(* CODESYS project uninc.library
   Company: Beckhoff Automation GmbH & Co. KG
   DefaultNamespace: TC3_UniNC
   Version: 1.0.6.2
   Placeholder: UniNc Gruppe 11
   Author: Bernhard Edenfeld, Benedikt Daut, Christian Frickenstein
   Description: FBs für die Nutzung der NC, Sercos-Achsen, Encoder-Achsen und Eil-Schleichachsen im Stil der Gruppe 11
   Title: UniNc Gruppe 11

Project tree, tasks and I/O mapping:
  libraries: Tc2_MC2, * (Beckhoff Automation GmbH); Tc2_MC2_Drive, * (Beckhoff Automation GmbH); Tc2_Standard, * (Beckhoff Automation GmbH); Tc2_System, * (Beckhoff Automation GmbH); UniLib Gruppe 11, * (Beckhoff Automation GmbH & Co. KG)
  DUTs/
    data type E_AchsFahrauftraege
    data type ST_DiagAxis
    data type ST_UniEinschleifen
  GVLs/
    global variables GlobalVar_NC
    global variables NcParameter
  POUs/
    function block FB_AchsKontrlAnstg [ST]: a_AchsStatus, b_AchsParam, c_AchsFreigb, d_AchsReferz, e_AchsHdFkt, f_AchsKopplg, g_AchsAuftrg, h_AchsEndlos, i_AchsModulo, k_AchsReset, x_AchsMeldg
    function block FB_AchsStartAusf [ST]
    function block FB_Bremsentest_BremseEinschleifen [ST]: a_Error, a_LogZeile, b_AnwEinschleifen
    function block FB_BremsentestMitLog [ST]: a_Error, a_LogZeile
    function block FB_BremsentestMitLog_FW07 [ST]: a_Error, a_LogZeile
    function block FB_CtrlXGrupEinschalt [ST]
  VISUs/
    Intern/
      visualisation V_DiagAchse
  text list GlobalTextList
*)

// DUTs/E_AchsFahrauftraege
{attribute 'qualified_only'}
{attribute 'strict'}
TYPE E_AchsFahrauftraege :
(
	eKoppelPosition 			:= 1,	// Index für arrPTP_start[]: Achse fährt eine Korrekturposition an um mit einer Masterachse zu koppeln mit 5% der Max-Geschwindigkeit
	eGrundPosition				:= 2,	// Index für arrPTP_start[]: Achse fährt die Grundposition aus den Parametern an mit 25% der Max-Geschwindigkeit
	eBearbeitungsPosition	:= 3	// Index für arrPTP_start[]: Achse fährt zur Bearbeitungsposition aus den Zielvorgaben an mit der prozentual gewählten Zielgeschwindigkeit
);
END_TYPE

// DUTs/ST_DiagAxis
TYPE ST_DiagAxis :
STRUCT
	nAcutalLength	: UINT;	// Tatsächliche länge der Meldung
	nMaxLength		: UINT;	// Maximal mögliche länge der Meldung 
	sDiagMessage	: T_MaxString;	// Standardlänge der Meldung. Kann aber beschränkt ausgelesen werden durch nAcutalLength.
END_STRUCT
END_TYPE

// DUTs/ST_UniEinschleifen
// Struktur für eine standardisierte Grundstellungsanwahl mit einer HMI-Taste und Meldungen 
{attribute 'pack_mode' := '1'}
TYPE ST_UniEinschleifen :
STRUCT
// Eine Handfunktionstaste für die Grundstellungsfahrt.
{attribute 'MaschPara.Name' := 'Handfunktion:'}	// Das Array ist Teil der Handfunktionen und wird mit 'Handfunktion:' betitelt
{attribute 'MaschPara.Handfunktion.Btn1' := '1 TextHandFkt'} // Handfunktion.Btn[X] ist der Taster im Array. TextHandFkt ist default Text, wenn z.B. die PLC nicht läuft
	stHandFktHMI		: ARRAY [1..1] OF ST_HandFktHMI;

END_STRUCT
END_TYPE

// GVLs/GlobalVar_NC
{attribute 'Tc2GvlVarNames'}
VAR_GLOBAL
	arrStartAusf							:ARRAY[0..cAnzAchsen] OF FB_AchsStartAusf;	// Vorschlag für eine allgemeine Instanz: Achsstart-FB für alle Achsen vordefiniert. Kann im Projekt aufgerufen werden. 

	arrNcAchsReset							:ARRAY[0..cAnzAchsen] OF BOOL;	// Vorschlag für eine allgemeine Variable: NC-AchsReset für eine bestimmte Achse 
	
	arrAchsDiag								:ARRAY[0..cAnzAchsen] OF Tc2_System.T_MaxString;	// Diagnose/Zustand der SoE-Achsen. S-0-0095
	
	// Allgemeine Achsvariablen
	bNcAchsResetErfordl					:BOOL;	// Vorschlag für eine allgemeine Variable: mindestens eine NC-Achse hat einen Fehler und ein Reset ist erforderlich.
	bAchsFreifahrErfordl					:BOOL;	// Vorschlag für eine allgemeine Variable: mindestens eine Achse hat oder hatte die Endlagen angefahren und muss von dieser manuell heruntergefahren werden
	bAchsRestartErfordl					:BOOL;	// Vorschlag für eine allgemeine Variable:
	bNcAchsResetAngw						:BOOL;	// Vorschlag für eine allgemeine Variable: NC-Reset wurde durch Bediener angewählt
	bAchsFreifahrAngw						:BOOL;	// Vorschlag für eine allgemeine Variable: Achsen Freifahren wurde durch Bediener angewählt
	bAntriebResetAktiv					:BOOL;	// Vorschlag für eine allgemeine Variable: Hardware-Reset ist aktiv
	
	// Override
	fOverridePTP							:LREAL:= 100;	// Vordefinierter maximaler Override für alle Achsen
END_VAR
VAR_GLOBAL CONSTANT
	// Fahraufträge Achsen
	cKopplPos	: INT:= 1;	// Index für arrPTP_start[]: Achse fährt eine Korrekturposition an um mit einer Masterachse zu koppeln mit 5% der Max-Geschwindigkeit
	cGrundPos	: INT:= 2;	// Index für arrPTP_start[]: Achse fährt die Grundposition aus den Parametern an mit 25% der Max-Geschwindigkeit
	cBearbPos	: INT:= 3;	// Index für arrPTP_start[]: Achse fährt zur Bearbeitungsposition aus den Zielvorgaben an mit der prozentual gewählten Zielgeschwindigkeit
END_VAR

// GVLs/NcParameter
{attribute 'Tc2GvlVarNames'}
VAR_GLOBAL CONSTANT
	// Gesamtanzahl Achsen
	cAnzAchsen			: INT:= 100;	// Achsen mit Encoder und Drive. Also auch Eil-Schleichachsen und Encoderachsen
	cAnzAchsenReal		: INT:= 8;	// Nur Achsen mit Drive. Also SoE und Eil-Schleichachsen
END_VAR

// POUs/FB_AchsKontrlAnstg
(*
Beschreibung :	Allg. Achshändling (MC2-Lib)
					Datentypen: Struct_NcAchsen
TwinCat Vers.:	3.1.4024.25							
Erstellt		 :	Anlagentechnik Grp.11 (BECKHOFF AUTOMATION)
*)
FUNCTION_BLOCK FB_AchsKontrlAnstg
VAR_IN_OUT
	IQ_stAchse						: TC3_UniLib.ST_NcAchsen;
	IQ_fbAxisRef					: Tc2_MC2.AXIS_REF;
END_VAR
VAR_INPUT
	I_refNcAchsen					: REFERENCE TO ARRAY [1..cAnzAchsen] OF Tc2_MC2.AXIS_REF;
	I_nBetrArt						: INT	:= 0;		(*0:Standard-PTP/1:Endlosbetrieb/2:Modulobetrieb *)
	I_fOverride						: LREAL := 100;	// Override für diese Achse, bei Nichtverwendung 100%
	I_bEndlagenExtern				: BOOL;
	I_bAutoStopAktiv				: BOOL := TRUE;
{attribute 'hide'}	
	I_eRichtungModulo				: MC_Direction := MC_Positive_Direction;
END_VAR
VAR_OUTPUT
END_VAR
VAR
	(*a_AchsStatus*)
	tonHwFehler			:Tc2_Standard.TON;
	stDiagAxis			:ST_DiagAxis;
	nIdn					:WORD;

	(*b_AchsParam*)
	fbAchsPar1L			:Tc2_MC2.MC_ReadParameter;
	stAchsPar1LOut		:Tc2_MC2.ST_McOutputs;
	fbAchsPar2L			:Tc2_MC2.MC_ReadParameter;
	stAchsPar2LOut		:Tc2_MC2.ST_McOutputs;
	fbAchsPar3L			:Tc2_MC2.MC_ReadBoolParameter;
	stAchsPar3LOut		:Tc2_MC2.ST_McOutputs;
	fbAchsPar4L			:Tc2_MC2.MC_ReadBoolParameter;
	stAchsPar4LOut		:Tc2_MC2.ST_McOutputs;
	fbAchsPar5L			:Tc2_MC2.MC_ReadParameter;
	stAchsPar5LOut		:Tc2_MC2.ST_McOutputs;
	fbAchsPar1S			:Tc2_MC2.MC_WriteParameter;
	stAchsPar1SOut		:Tc2_MC2.ST_McOutputs;
	fbAchsPar2S			:Tc2_MC2.MC_WriteParameter;
	stAchsPar2SOut		:Tc2_MC2.ST_McOutputs;
	
	fbAchsParName		:Tc2_MC2.MC_ReadParameterSet;
	stAchsParSet		:Tc2_MC2.ST_AxisParameterSet;
	stAchsParName		:Tc2_MC2.ST_McOutputs;

	rtrigParamLesZykl	:Tc2_Standard.R_TRIG;
	bEndlMinLes			:BOOL;
	bEndlMinSchr		:BOOL;
	fEndlBegrMin		:LREAL;
	bEndlMaxLes			:BOOL;
	bEndlMaxSchr		:BOOL;
	fEndlBegrMax		:LREAL;

	(*c_AchsFreigb*)
	fbAchsFreig			:Tc2_MC2.MC_Power;
	stAchsFreigOut		:Tc2_MC2.ST_McOutputs;

	tonVerzVorschFrg	:Tc2_Standard.TON;
	tonVerzEndlgStop	:Tc2_Standard.TON;
	tonVerzAntrbFehl	:Tc2_Standard.TON;

	(*d_AchsReferz*)
	fbAchsReferenz		:Tc2_MC2.MC_Home;
	stAchsReferenzOut	:Tc2_MC2.ST_McOutputs;
	fbAchsIstwSetz		:Tc2_MC2.MC_SetPosition;
	stAchsIstwSetzOut	:Tc2_MC2.ST_McOutputs;

	(*e_AchsHdFkt*)
	fbAchsHandfkt		:Tc2_MC2.MC_Jog;
	stAchsHandfktOut	:Tc2_MC2.ST_McOutputs;

	(*f_AchsKopplg*)
	fbAchsAnkoppln		:Tc2_MC2.MC_GearInDyn;
	stAchsAnkopplnOut	:Tc2_MC2.ST_McOutputs;
	fbAchsAbkoppln		:Tc2_MC2.MC_GearOut;
	stAchsAbkopplnOut	:Tc2_MC2.ST_McOutputs;

	(*g_AchsAuftrg*)
	fbAchsStartA1		:Tc2_MC2.MC_MoveAbsolute; (*Standard*)
	fbAchsStartA2		:Tc2_MC2.MC_MoveVelocity; (*Endlos*)
	fbAchsStartA3		:Tc2_MC2.MC_MoveModulo; (*Modulo*)
	stAchsStartAOut	:Tc2_MC2.ST_McOutputs;
	fbAchsStartB1		:Tc2_MC2.MC_MoveAbsolute; (*Standard*)
	fbAchsStartB2		:Tc2_MC2.MC_MoveVelocity; (*Endlos*)
	fbAchsStartB3		:Tc2_MC2.MC_MoveModulo; (*Modulo*)
	stAchsStartBOut	:Tc2_MC2.ST_McOutputs;
	fbAchsStop			:Tc2_MC2.MC_Halt;
	stAchsStopOut		:Tc2_MC2.ST_McOutputs;

	fAuftrZielPos		:LREAL;
	fLetztZielPos		:LREAL;
	fAuftrGeschw		:LREAL;
	fLetztGeschw		:LREAL;
	nAuftrBuffMode		:Tc2_MC2.MC_BufferMode;
	bAuftrStart			:BOOL;
	nAuftrState			:INT;
	bNeuAuftrVorg		:BOOL;
	bAuftrStartA		:BOOL;
	bAuftrAktivA		:BOOL;
	bAuftrFertigA		:BOOL;
	bAuftrStartB		:BOOL;
	bAuftrAktivB		:BOOL;
	bAuftrFertigB		:BOOL;
	bAuftrStop			:BOOL;
	bAuftrGestoppt		:BOOL;
	fAuftrOverride		:LREAL;
	tonAuftrLfZeit		:Tc2_Standard.TON;

	(*k_AchsReset*)
	tpReset				:Tc2_Standard.TP;
	bInit					:BOOL;
	fbAchsReset			:Tc2_MC2.MC_Reset;
	stAchsResetOut		:Tc2_MC2.ST_McOutputs;

	(*x_AchsMeldg*)
	nAchsMeldNr			:INT;
	fbDiagMessages		:FB_SoERead;
END_VAR

	(*Achs-Kontrollfkt./-Ansteuerung*)
	
	(**************************************************)	

	a_AchsStatus();	(*Achsstatus lesen/sotieren*)
							(*Achsenistwert lesen*)

	(**************************************************)	

	b_AchsParam();		(*Achsparameter lesen*)
							(*Achsparameter schreiben*)

	(**************************************************)	

	c_AchsFreigb();	(*Achsfreigaben ermitteln*)
							(*Achsfreigaben schreiben*)

	(**************************************************)	

	d_AchsReferz();	(*Achse referieren*)
							(*Achsistwert setzen*)

	(**************************************************)	

	e_AchsHdFkt();		(*Achshandfunktionen*)

	(**************************************************)	

	f_AchsKopplg();	(*Achse an.-abkoppeln*)

	(**************************************************)	

	CASE I_nBetrArt OF
0:	g_AchsAuftrg();	(*Achswerte schreiben / Achse starten / Achse stoppen*)
1:	h_AchsEndlos();	(*			0:Standard-PTP / 1:Endlosbetrieb /2:Modulobetrieb            *)
2:	i_AchsModulo();	(*			0:Standard-PTP / 1:Endlosbetrieb /2:Modulobetrieb            *)
	END_CASE

	(**************************************************)	

	k_AchsReset();		(*Achse zurücksetzen*)

	(**************************************************)	

	x_AchsMeldg();		(*Achsmeldungen ausgeben*)

	(**************************************************)

ACTION a_AchsStatus:
	// Achsstatus lesen/sotieren
	IQ_fbAxisRef.ReadStatus();
	IQ_stAchse.nAxNr						:= TO_INT(IQ_fbAxisRef.NcToPlc.AxisId);

	IQ_stAchse.bNcFehler					:= IQ_fbAxisRef.Status.Error;
	IQ_stAchse.nFehlerNr					:= IQ_fbAxisRef.Status.ErrorID;
	IQ_stAchse.bBetrbBer					:= IQ_fbAxisRef.Status.Operational;

	IQ_stAchse.stStatus.bInReferz		:= IQ_fbAxisRef.Status.Homed;
	IQ_stAchse.stStatus.bInStillst	:= IQ_fbAxisRef.Status.NotMoving;
	IQ_stAchse.stStatus.bFahrbewAkt	:= IQ_fbAxisRef.Status.Moving;
	IQ_stAchse.stStatus.bFaehrtPos	:= IQ_fbAxisRef.Status.PositiveDirection;
	IQ_stAchse.stStatus.bFaehrtNeg	:= IQ_fbAxisRef.Status.NegativeDirection;
	IQ_stAchse.stStatus.bKonstFahrt	:= IQ_fbAxisRef.Status.ConstantVelocity;
	IQ_stAchse.stStatus.bZielPosErr	:= IQ_fbAxisRef.Status.InTargetPosition;
	IQ_stAchse.stStatus.bZielBerErr	:= IQ_fbAxisRef.Status.InPositionArea;
	// Struktur eventuell erweitern
	
	// Hardwarefehler
	tonHwFehler(
		IN:= (( (NOT IQ_stAchse.stStatus.bAchseBTB
						OR NOT IQ_stAchse.bBetrbBer	)
					AND IQ_stAchse.stStatus.bFrgSchutzBer)
				OR (IQ_fbAxisRef.Status.Error
					AND IQ_fbAxisRef.Status.ErrorID = 18000)),
		PT:= t#5s);
		
	IQ_stAchse.bHwFehler	:= tonHwFehler.Q;

	// Achsenistwert lesen
	IQ_stAchse.fPosIstwert				:= IQ_fbAxisRef.NcToPlc.ActPos;
	IQ_stAchse.fVeloIstwert				:= IQ_fbAxisRef.NcToPlc.ActVelo;
	IQ_stAchse.fModIstwert				:= IQ_fbAxisRef.NcToPlc.ModuloActPos;

	// Bereichsmeldung Istwert
	IF IQ_stAchse.stStatus.bInReferz
		AND IQ_stAchse.stParam.bSoftEndlAkt
		AND ((IQ_stAchse.fPosIstwert + 5) < IQ_stAchse.stParam.fSoftEndlMin
		OR   (IQ_stAchse.fPosIstwert - 5) > IQ_stAchse.stParam.fSoftEndlMax)
		THEN
			IQ_stAchse.stMeldg.bIstPosFehl:= TRUE;
		ELSE
			IQ_stAchse.stMeldg.bIstPosFehl:= FALSE;
	END_IF

	// S-0-0095 Meldungen auslesen
	nIdn :=  S_0_IDNs +95;
	
	fbDiagMessages(
		NetId		:= IQ_fbAxisRef.ADS.NetId,	// Hier die Net-Id aus der Achsstrukur nehmen. Für den Fall, dass die Achse in einem Anderen Zielsystem läuft
		Idn		:= nIdn, 
		Element	:= 16#40, 
		pDstBuf	:= ADR(stDiagAxis), 
		BufLen	:= SIZEOF(stDiagAxis), 
		Execute	:= bTaktLangsam, 
		Timeout	:= t#5s, 
		Axis		:= IQ_fbAxisRef);

	IF IQ_stAchse.nAxNr > cAnzAchsen
	THEN
		arrAchsDiag[0] := CONCAT('AchsID: ',
								CONCAT(TO_STRING(IQ_stAchse.nAxNr),
								CONCAT(' ist höher als cAnzAchsen. ',
									DELETE(stDiagAxis.sDiagMessage,
										TO_INT(SIZEOF(T_MAXSTRING)-stDiagAxis.nAcutalLength),
										TO_INT(stDiagAxis.nAcutalLength)))));
	ELSIF NOT fbDiagMessages.Busy
		AND fbDiagMessages.Error
	THEN
		arrAchsDiag[IQ_stAchse.nAxNr] := '';
		arrAchsDiag[IQ_stAchse.nAxNr] := stDiagAxis.sDiagMessage;
		arrAchsDiag[IQ_stAchse.nAxNr] := DELETE(arrAchsDiag[IQ_stAchse.nAxNr],
													TO_INT(SIZEOF(T_MAXSTRING)-stDiagAxis.nAcutalLength),
													TO_INT(stDiagAxis.nAcutalLength));
	
	ELSIF fbDiagMessages.Error
	THEN
		arrAchsDiag[IQ_stAchse.nAxNr] := 'ADS-Error: ';
		arrAchsDiag[IQ_stAchse.nAxNr] := CONCAT(arrAchsDiag[IQ_stAchse.nAxNr],F_AdsErrorIdToString(fbDiagMessages.AdsErrId));
		arrAchsDiag[IQ_stAchse.nAxNr] := CONCAT(arrAchsDiag[IQ_stAchse.nAxNr],' Sercos-Error: ');
		arrAchsDiag[IQ_stAchse.nAxNr] := CONCAT(arrAchsDiag[IQ_stAchse.nAxNr],TO_STRING(fbDiagMessages.SercosErrId));
	END_IF

// ENDE
END_ACTION

ACTION b_AchsParam:
// Achsparameter lesen
rtrigParamLesZykl (CLK:= IQ_stAchse.stParam.bLesSchrFrg);

fbAchsPar1L (Axis					:= IQ_fbAxisRef,	(*Softendlage Min. /Wert*)
				 Enable				:= rtrigParamLesZykl.Q
											OR bEndlMinLes,
				 ParameterNumber	:= AxisMinSoftPosLimit,
				 ReadMode			:= ReadMode_Once,

				 Busy					=>	stAchsPar1LOut.Busy,
				 Error				=>	stAchsPar1LOut.Error,
				 ErrorID				=>	stAchsPar1LOut.ErrorID);

fbAchsPar2L (Axis					:= IQ_fbAxisRef,	(*Softendlage Max. /Wert*)
				 Enable				:= rtrigParamLesZykl.Q
											OR bEndlMaxLes,
				 ParameterNumber	:= AxisMaxSoftPosLimit,
				 ReadMode			:= ReadMode_Once,

				 Busy					=>	stAchsPar2LOut.Busy,
				 Error				=>	stAchsPar2LOut.Error,
				 ErrorID				=>	stAchsPar2LOut.ErrorID);

fbAchsPar3L (Axis					:= IQ_fbAxisRef,	(*Softendlage Min. aktiv*)
				 Enable				:= rtrigParamLesZykl.Q,
				 ParameterNumber	:= AxisEnMinSoftPosLimit,
				 ReadMode			:= ReadMode_Once,

				 Busy					=>	stAchsPar3LOut.Busy,
				 Error				=>	stAchsPar3LOut.Error,
				 ErrorID				=>	stAchsPar3LOut.ErrorID);

fbAchsPar4L (Axis					:= IQ_fbAxisRef,	(*Softendlage Max. aktiv*)
				 Enable				:= rtrigParamLesZykl.Q,
				 ParameterNumber	:= AxisEnMaxSoftPosLimit,
				 ReadMode			:= ReadMode_Once,

				 Busy					=>	stAchsPar4LOut.Busy,
				 Error				=>	stAchsPar4LOut.Error,
				 ErrorID				=>	stAchsPar4LOut.ErrorID);

// Alle Achsparameter auslesen, damit wird auch der Achsname ausgelesen
fbAchsParName(
	Axis					:= IQ_fbAxisRef, 
	Execute				:= rtrigParamLesZykl.Q,
	Parameter			:= stAchsParSet, 
	
	Done					=> stAchsParName.Done, 
	Busy					=> stAchsParName.Busy, 
	Error					=> stAchsParName.Error, 
	ErrorID				=> stAchsParName.ErrorID
);

IF stAchsParName.Done
THEN
	IQ_stAchse.sAxName	:= stAchsParSet.sAxisName;
END_IF

IF fbAchsPar1L.Valid
	THEN
		IQ_stAchse.stParam.fSoftEndlMin:= fbAchsPar1L.Value;
END_IF

IF fbAchsPar2L.Valid
	THEN
		IQ_stAchse.stParam.fSoftEndlMax:= fbAchsPar2L.Value;
END_IF

IF fbAchsPar3L.Valid AND fbAchsPar4L.Valid
	THEN
		IQ_stAchse.stParam.bSoftEndlAkt:= fbAchsPar3L.Value AND fbAchsPar4L.Value;
END_IF

// Eilganggeschwindigkeit auslesen
fbAchsPar5L (Axis					:= IQ_fbAxisRef,
				 Enable				:= rtrigParamLesZykl.Q,
				 ParameterNumber	:= AxisMaxVelocity,
				 ReadMode			:= ReadMode_Once,

				 Busy					=>	stAchsPar5LOut.Busy,
				 Error				=>	stAchsPar5LOut.Error,
				 ErrorID				=>	stAchsPar5LOut.ErrorID);

IF fbAchsPar5L.Valid
	THEN
		IQ_stAchse.stParam.fEilgGeschw:= fbAchsPar5L.Value;
END_IF

// Achsparameter schreiben
IF bEndlMinSchr
	THEN
		bEndlMinLes:= TRUE;
		bEndlMinSchr:= FALSE;
	ELSE
		bEndlMinLes:= FALSE;
END_IF

IF IQ_stAchse.stParam.fEndlBegrMin <> fEndlBegrMin
	AND NOT bEndlMinLes
	AND NOT bEndlMinSchr
	AND IQ_stAchse.stParam.bLesSchrFrg
	THEN
		fEndlBegrMin:= IQ_stAchse.stParam.fEndlBegrMin;
		bEndlMinSchr:= TRUE;
END_IF

IF bEndlMaxSchr
	THEN
		bEndlMaxLes:= TRUE;
		bEndlMaxSchr:= FALSE;
	ELSE
		bEndlMaxLes:= FALSE;
END_IF

IF IQ_stAchse.stParam.fEndlBegrMax <> fEndlBegrMax
	AND NOT bEndlMaxLes
	AND NOT bEndlMaxSchr
	AND IQ_stAchse.stParam.bLesSchrFrg
	THEN
		fEndlBegrMax:= IQ_stAchse.stParam.fEndlBegrMax;
		bEndlMaxSchr:= TRUE;
END_IF

// Softwareendlage Minimum schreiben
fbAchsPar1S (Axis					:= IQ_fbAxisRef,	(*Softendlage Min. /Wert*)
				 Execute				:= bEndlMinSchr,
				 ParameterNumber	:= AxisMinSoftPosLimit,
				 Value				:= fEndlBegrMin,

				 Busy					=>	stAchsPar1SOut.Busy,
				 Error				=>	stAchsPar1SOut.Error,
				 ErrorID				=>	stAchsPar1SOut.ErrorID);

// Softwareendlage Maximum schreiben
fbAchsPar2S (Axis					:= IQ_fbAxisRef,	(*Softendlage Max. /Wert*)
				 Execute				:= bEndlMaxSchr,
				 ParameterNumber	:= AxisMaxSoftPosLimit,
				 Value				:= fEndlBegrMax,

				 Busy					=>	stAchsPar2SOut.Busy,
				 Error				=>	stAchsPar2SOut.Error,
				 ErrorID				=>	stAchsPar2SOut.ErrorID);
END_ACTION

ACTION c_AchsFreigb:
	(*Achsfreigaben ermitteln*)
	IF NOT I_bEndlagenExtern
		AND NOT IQ_stAchse.stParam.bOhnSoftEndl
	THEN
		IQ_stAchse.stFreigb.bSensEndlPos	:= IQ_stAchse.stEinAusG.I_nDigitaleEingaenge.3;
		IQ_stAchse.stFreigb.bSensEndlNeg	:= IQ_stAchse.stEinAusG.I_nDigitaleEingaenge.4;
	END_IF

	IF IQ_stAchse.stFreigb.bAntrbEinFrg
		AND NOT IQ_stAchse.bNcFehler
		THEN
			IQ_stAchse.stFreigb.bReglerFrg:= TRUE;
		ELSE
			IQ_stAchse.stFreigb.bReglerFrg:= FALSE;
	END_IF


	IF NOT IQ_stAchse.stFreigb.bSensEndlNeg
		THEN
			IF IQ_stAchse.stFreigb.bAntrbEinFrg
				THEN
					IQ_stAchse.stMeldg.bEndlNegAngf:= TRUE;
			END_IF
		ELSE
			IF IQ_stAchse.stFreigb.bEndlFreifAkt
				THEN
					IQ_stAchse.stMeldg.bEndlNegAngf:= FALSE;
			END_IF
	END_IF

	IF NOT IQ_stAchse.stFreigb.bSensEndlPos
		THEN
			IF IQ_stAchse.stFreigb.bAntrbEinFrg
				THEN
					IQ_stAchse.stMeldg.bEndlPosAngf:= TRUE;
			END_IF
		ELSE
			IF IQ_stAchse.stFreigb.bEndlFreifAkt
				THEN
					IQ_stAchse.stMeldg.bEndlPosAngf:= FALSE;
			END_IF
	END_IF


	tonVerzVorschFrg (IN:= IQ_stAchse.bBetrbBer
							  	  AND IQ_stAchse.stFreigb.bReglerFrg
							     AND IQ_stAchse.stFreigb.bVorschFrg
							     AND (IQ_stAchse.stFreigb.bEndlFreifAkt
							     OR NOT IQ_stAchse.stMeldg.bEndlNegAngf)
							     AND (IQ_stAchse.stFreigb.bEndlFreifAkt
							     OR NOT IQ_stAchse.stMeldg.bEndlPosAngf),
						   PT:= T#150MS);

	IQ_stAchse.stFreigb.bVorsFrgNeg:= NOT IQ_stAchse.stMeldg.bEndlNegAngf
													 		 	 AND tonVerzVorschFrg.Q;
	IQ_stAchse.stFreigb.bVorsFrgPos:= NOT IQ_stAchse.stMeldg.bEndlPosAngf
													 		 	 AND tonVerzVorschFrg.Q;


	tonVerzEndlgStop (IN:= IQ_stAchse.stMeldg.bEndlNegAngf
							     OR IQ_stAchse.stMeldg.bEndlPosAngf,
						   PT:= T#500MS);

	IQ_stAchse.stFreigb.bEndlgStop:= NOT IQ_stAchse.stFreigb.bEndlFreifAkt
															   AND tonVerzEndlgStop.Q;

	// Für die NC und Beckhoff-Servos: Endlagen werden überschrieben
	IQ_fbAxisRef.PlcToNc.ControlDWord.8:= IQ_stAchse.stFreigb.bEndlFreifAkt;

	(*Achsfreigaben schreiben*)

	fbAchsFreig (Axis			   	:= IQ_fbAxisRef,
				    Enable				:=	IQ_stAchse.stFreigb.bReglerFrg,
				    Enable_Positive	:=	IQ_stAchse.stFreigb.bVorsFrgPos,
				    Enable_Negative	:=	IQ_stAchse.stFreigb.bVorsFrgNeg,
				    Override			:= fAuftrOverride,
				    BufferMode			:= MC_Aborting,

				    Busy					=>	stAchsFreigOut.Busy,
				    Error				=>	stAchsFreigOut.Error,
				    ErrorID				=>	stAchsFreigOut.ErrorID);
					 
	IQ_stAchse.fAuftrOverride	:= fAuftrOverride;	// Internen Override in die Achsstruktur schieben

	(*Meldung Antriebsüberwachung*)

	tonVerzAntrbFehl (IN:= IQ_stAchse.stFreigb.bReglerFrg
							     AND NOT IQ_stAchse.bBetrbBer,
						   PT:= T#5S);

	IQ_stAchse.stMeldg.bAntrbFehl:= tonVerzAntrbFehl.Q;
END_ACTION

ACTION d_AchsReferz:
// Referenzsensor zuweisen
IQ_fbAxisRef.PlcToNc.ControlDWord.5	:= IQ_stAchse.stGrdfkt.bRefrzSensor;

// Achse referieren

	fbAchsReferenz (Axis					:= IQ_fbAxisRef,
					    Execute				:= IQ_stAchse.stGrdfkt.bRefrz_ausf
													AND IQ_stAchse.stFreigb.bVorsFrgNeg
													AND IQ_stAchse.stFreigb.bVorsFrgPos,
					    Position			:= DEFAULT_HOME_POSITION,
					    HomingMode			:= MC_DefaultHoming,
					    BufferMode			:= MC_Aborting,
					    bCalibrationCam	:= IQ_stAchse.stGrdfkt.bRefrzSensor,

					    Done					=> IQ_stAchse.stGrdfkt.bRefrz_ausgf,

				  	    Busy					=>	stAchsReferenzOut.Busy,
				       Error				=>	stAchsReferenzOut.Error,
				       ErrorID				=>	stAchsReferenzOut.ErrorID);

	(*Achsistwert setzen*)

	fbAchsIstwSetz (Axis					:= IQ_fbAxisRef,
					    Execute				:= IQ_stAchse.stGrdfkt.bIstw_setz,
					    Position			:= IQ_stAchse.stGrdfkt.fIstSetzwert,
					    Mode					:= FALSE, (*Absolut*)

					    Done					=> IQ_stAchse.stGrdfkt.bIstw_gesetz,

				  	    Busy					=>	stAchsIstwSetzOut.Busy,
				       Error				=>	stAchsIstwSetzOut.Error,
				       ErrorID				=>	stAchsIstwSetzOut.ErrorID);
END_ACTION

ACTION e_AchsHdFkt:
	(*Achshandfunktionen*)

	fbAchsHandfkt (Axis				:= IQ_fbAxisRef,
					   JogForward 		:= IQ_stAchse.stGrdfkt.bHdfkt_pos
										   	AND IQ_stAchse.stFreigb.bVorsFrgPos,
					   JogBackwards 	:= IQ_stAchse.stGrdfkt.bHdfkt_neg
												AND IQ_stAchse.stFreigb.bVorsFrgNeg,
					   Mode				:= MC_Jogmode_Standard_Slow,
					   Position 		:= 0,	(*SystemManager*)
					   Velocity			:= 0,	(*SystemManager*)
					   Acceleration	:= 0,	(*SystemManager*)
					   Deceleration	:= 0,	(*SystemManager*)
					   Jerk				:= 0,	(*SystemManager*)

				      Busy				=>	stAchsHandfktOut.Busy,
				      Error				=>	stAchsHandfktOut.Error,
				      ErrorID			=>	stAchsHandfktOut.ErrorID);
END_ACTION

ACTION f_AchsKopplg:
	(*Achse an.-abkoppeln*)

IF __ISVALIDREF(I_refNcAchsen)	// Hier muss abgefragt werden, ob die Referenz beschrieben wurde, sonst gibt es Page-Fault-Fehler
	AND IQ_stAchse.stKoppln.nKopplMaster <> IQ_stAchse.nAxNr	// wenn diese Achse der Master ist, muss nix gekoppelt werden. 
THEN
	CASE IQ_stAchse.stKoppln.nKopplMaster OF 1..cAnzAchsen:

	fbAchsAnkoppln (Master			:= I_refNcAchsen[IQ_stAchse.stKoppln.nKopplMaster],
					    Slave			:= IQ_fbAxisRef,
					    Enable			:= IQ_stAchse.stKoppln.bAnkoppln
										   	AND IQ_stAchse.stAuftrg.bPTP_PosiFrg,
					    GearRatio		:= IQ_stAchse.stKoppln.fKopplFakt,
					    Acceleration	:= 0,	(*SystemManager*)
				       Deceleration	:= 0,	(*SystemManager*)
				       Jerk				:= 0,	(*SystemManager*)
					    BufferMode		:= MC_Aborting,

					    InGear			=> IQ_stAchse.stKoppln.bAngekoplt,

					    Busy				=>	stAchsAnkopplnOut.Busy,
					    Error			=>	stAchsAnkopplnOut.Error,
					    ErrorID			=>	stAchsAnkopplnOut.ErrorID);

	END_CASE
END_IF

	fbAchsAbkoppln (Slave			:= IQ_fbAxisRef,
					    Execute			:= IQ_stAchse.stKoppln.bAbkoppln
										   	(*AND I_RefAchse.Auftrg.PTP_PosiFrg*),

					    Done				=> IQ_stAchse.stKoppln.bAbgekoplt,

					    Busy				=>	stAchsAbkopplnOut.Busy,
					    Error			=>	stAchsAbkopplnOut.Error,
					    ErrorID			=>	stAchsAbkopplnOut.ErrorID);

	IQ_stAchse.stKoppln.nKopplStat:= IQ_fbAxisRef.NcToPlc.CoupleState;
END_ACTION

ACTION g_AchsAuftrg:
	(*Achswerte schreiben / Achse starten / Achse stoppen*)
	(*-Standardachse*)

	IQ_stAchse.stAuftrg.sPTP_AuftrgTyp:= 'Standardachse';

	(*Achs-Fahrauftrag auswerten*)

	IF IQ_stAchse.stAuftrg.arrPTP_start[cKopplPos]		(*Korrekt-Koppelposition*)
		THEN
			fAuftrZielPos	:= IQ_stAchse.stKoppln.fKorrektPos;
			fAuftrGeschw	:= IQ_stAchse.stParam.fEilgGeschw * 0.05;
	ELSIF IQ_stAchse.stAuftrg.arrPTP_start[cGrundPos]	(*Grundstellungsposition*)
		THEN
			fAuftrZielPos	:= IQ_stAchse.stParam.fGrdstlgPos;
			fAuftrGeschw	:= IQ_stAchse.stParam.fEilgGeschw * 0.25;
	ELSIF IQ_stAchse.stAuftrg.arrPTP_start[cBearbPos]	(*Bearbeitungsposition*)
		THEN
			fAuftrZielPos	:= IQ_stAchse.stAuftrg.fPTP_ZielPos
									+ IQ_stAchse.stParam.fPosVerrWert
									+ IQ_stAchse.stParam.fPosOffsWert;
			fAuftrGeschw	:= (IQ_stAchse.stParam.fEilgGeschw / 100)
   								 * IQ_stAchse.stAuftrg.fPTP_Geschw;
	END_IF

	(*Achs-Fahrauftrag prüfen/starten*)

	IF IQ_stAchse.stAuftrg.arrPTP_start[cKopplPos]
		OR IQ_stAchse.stAuftrg.arrPTP_start[cGrundPos]
		OR IQ_stAchse.stAuftrg.arrPTP_start[cBearbPos]
		THEN
			IF (IQ_stAchse.stParam.bSoftEndlAkt
				AND fAuftrZielPos >= IQ_stAchse.stParam.fSoftEndlMin
				AND fAuftrZielPos <= IQ_stAchse.stParam.fSoftEndlMax)
				OR IQ_stAchse.stParam.bOhnSoftEndl
				THEN
					IF NOT bAuftrStart
						OR bNeuAuftrVorg
						THEN
							IF NOT bAuftrStart
								THEN
									nAuftrBuffMode:= IQ_stAchse.stAuftrg.ePTP_BuffMode;
								ELSE
									nAuftrBuffMode:= MC_Aborting;
							END_IF
							IF NOT bAuftrStop
							THEN
								bAuftrStart:= TRUE;
							END_IF

							IF nAuftrState = 1
								THEN
									nAuftrState:= 2;
								ELSE
									nAuftrState:= 1;
							END_IF

							bNeuAuftrVorg:= FALSE;

							fLetztZielPos:= fAuftrZielPos;
							fLetztGeschw:= fAuftrGeschw;
						ELSE
							bNeuAuftrVorg:= (fAuftrZielPos <> fLetztZielPos
											 	 OR fAuftrGeschw <> fLetztGeschw)
												AND NOT bAuftrStop;
					END_IF
				ELSE
					bAuftrStart:= FALSE;
					bNeuAuftrVorg:= FALSE;
					IQ_stAchse.stMeldg.bZielPosFehl:= TRUE;
			END_IF
		ELSE
			bAuftrStart:= FALSE;
			bNeuAuftrVorg:= FALSE;
			IQ_stAchse.stMeldg.bZielPosFehl:= FALSE;
	END_IF

	CASE nAuftrState OF

1: (*AchsStart "A"*)

	IF bAuftrStart
		THEN
			bAuftrStartA:= TRUE;
			bAuftrStartB:= FALSE;
	ELSE
		bAuftrStartA:= FALSE;
		bAuftrStartB:= FALSE;
	END_IF

2: (*AchsStart "B"*)

	IF bAuftrStart
		THEN
			bAuftrStartA:= FALSE;
			bAuftrStartB:= TRUE;
	ELSE
		bAuftrStartA:= FALSE;
		bAuftrStartB:= FALSE;
	END_IF

	END_CASE

	// Achs-Fahrauftrag stoppen
	bAuftrStop	:= IQ_stAchse.stAuftrg.bPTP_stop
						OR (IQ_stAchse.stAuftrg.bPTP_AutoStop
							AND I_bAutoStopAktiv);

	// Achs-Fahrauftrag verzögern
	IF IQ_stAchse.stAuftrg.bPTP_verz
	THEN
		fAuftrOverride	:=
			MIN ( IQ_stAchse.stFreigb.fOverride,	// Override über die Achsstruktur
			MIN ( I_fOverride,	// Override über den Eingang am Achs-Baustein
					fOverridePTP));	// maximaler Override über die globale Variable
	ELSE
		fAuftrOverride	:=
			MIN(I_fOverride,
			fOverridePTP);	// maximaler Override über die globale Variable
	END_IF

	// Achs-Fahrauftrag anhalten
	IF IQ_stAchse.stAuftrg.bPTP_halt
		THEN
			fAuftrOverride:= 0;	// Override 0%
	END_IF

	//Achs-Fahrauftrag freigeben
	IF NOT bAuftrStart
		AND IQ_stAchse.bBetrbBer
		AND IQ_stAchse.stFreigb.bVorsFrgPos
		AND IQ_stAchse.stFreigb.bVorsFrgNeg
		THEN
			IQ_stAchse.stAuftrg.bPTP_PosiFrg:= TRUE;
		ELSE
			IQ_stAchse.stAuftrg.bPTP_PosiFrg:= FALSE;
	END_IF

	// Achs-Fahrauftrag ausführen
	fbAchsStartA1 (Axis				:= IQ_fbAxisRef,
				      Execute			:= bAuftrStartA,
				      Position			:= fAuftrZielPos,
				      Velocity			:= fAuftrGeschw,
				      Acceleration	:= 0,	(*SystemManager*)
				      Deceleration	:= 0,	(*SystemManager*)
				      Jerk				:= 0,	(*SystemManager*)
				      BufferMode		:= nAuftrBuffMode,

					   Active			=> bAuftrAktivA,
				      Done				=> bAuftrFertigA,

				      Busy				=>	stAchsStartAOut.Busy,
				      Error				=>	stAchsStartAOut.Error,
				      ErrorID			=>	stAchsStartAOut.ErrorID);

	fbAchsStartB1 (Axis				:= IQ_fbAxisRef,
				      Execute			:= bAuftrStartB,
				      Position			:= fAuftrZielPos,
				      Velocity			:= fAuftrGeschw,
				      Acceleration	:= 0,	(*SystemManager*)
				      Deceleration	:= 0,	(*SystemManager*)
				      Jerk				:= 0,	(*SystemManager*)
				      BufferMode		:= nAuftrBuffMode,

					   Active			=> bAuftrAktivB,
				      Done				=> bAuftrFertigB,

				      Busy				=>	stAchsStartBOut.Busy,
				      Error				=>	stAchsStartBOut.Error,
				      ErrorID			=>	stAchsStartBOut.ErrorID);

	fbAchsStop    (Axis				:= IQ_fbAxisRef,
				      Execute			:= bAuftrStop,
				      Deceleration	:= 0,	(*SystemManager*)
				      Jerk				:= 0,	(*SystemManager*)
				      BufferMode		:= MC_Aborting,

				      Done				=> bAuftrGestoppt,

				      Busy				=>	stAchsStopOut.Busy,
				      Error				=>	stAchsStopOut.Error,
				      ErrorID			=>	stAchsStopOut.ErrorID);


	IQ_stAchse.stAuftrg.fPTP_LetzZiel:= fLetztZielPos;

	IQ_stAchse.stAuftrg.bPTP_aktiv	:= (bAuftrStartA AND bAuftrAktivA)
										   		 		 		OR (bAuftrStartB AND bAuftrAktivB);
	IQ_stAchse.stAuftrg.bPTP_inZiel	:= (bAuftrStartA AND bAuftrFertigA)
										    		  		  		OR (bAuftrStartB AND bAuftrFertigB);
	IQ_stAchse.stAuftrg.bPTP_inFenst	:= IQ_stAchse.fPosIstwert < (fLetztZielPos + 0.1)
													  		  		AND IQ_stAchse.fPosIstwert > (fLetztZielPos - 0.1);
	IQ_stAchse.stAuftrg.bPTP_gest		:= bAuftrGestoppt;

	// Laufzeitmeldung Fahrauftrag
	tonAuftrLfZeit (IN:= bAuftrStart
							   AND NOT IQ_stAchse.stAuftrg.bPTP_stop
						      AND NOT IQ_stAchse.stAuftrg.bPTP_halt
						      AND NOT IQ_stAchse.stAuftrg.bPTP_inZiel,
					    PT:= T#60S);

	IQ_stAchse.stMeldg.bLfZeitFehl:= tonAuftrLfZeit.Q;
END_ACTION

ACTION h_AchsEndlos:
	(*Achswerte schreiben / Achse starten / Achse stoppen*)
	(*-Endlosachse*)

	IQ_stAchse.stAuftrg.sPTP_AuftrgTyp:= 'Endlosbetrieb';

	(*Achs-Fahrauftrag auswerten*)

	IF IQ_stAchse.stAuftrg.arrPTP_start[cBearbPos]	(*Bearbeitungsposition*)
		THEN
			fAuftrZielPos	:= IQ_stAchse.stAuftrg.fPTP_ZielPos;
			fAuftrGeschw	:= (IQ_stAchse.stParam.fEilgGeschw / 100)
   								 * IQ_stAchse.stAuftrg.fPTP_Geschw;
	END_IF

	(*Achs-Fahrauftrag prüfen/starten*)

	IF IQ_stAchse.stAuftrg.arrPTP_start[cBearbPos]
		THEN
			IF TRUE  (*Ohne Zielposvorgabe*)
				THEN
					IF NOT bAuftrStart
						OR bNeuAuftrVorg
						THEN
							IF NOT bAuftrStart
								THEN
									nAuftrBuffMode:= IQ_stAchse.stAuftrg.ePTP_BuffMode;
								ELSE
									nAuftrBuffMode:= MC_Aborting;
							END_IF

							IF NOT bAuftrStop
							THEN
								bAuftrStart:= TRUE;
							END_IF

							IF nAuftrState = 1
								THEN
									nAuftrState:= 2;
								ELSE
									nAuftrState:= 1;
							END_IF

							bNeuAuftrVorg:= FALSE;

							fLetztGeschw:= fAuftrGeschw;
						ELSE
							bNeuAuftrVorg:= (fAuftrGeschw <> fLetztGeschw)
													AND NOT bAuftrStop;
					END_IF
				ELSE
					bAuftrStart:= FALSE;
					bNeuAuftrVorg:= FALSE;
					IQ_stAchse.stMeldg.bZielPosFehl:= TRUE;
			END_IF
		ELSE
			bAuftrStart:= FALSE;
			bNeuAuftrVorg:= FALSE;
			IQ_stAchse.stMeldg.bZielPosFehl:= FALSE;
	END_IF

	CASE nAuftrState OF

1: (*AchsStart "A"*)

	IF bAuftrStart
		THEN
			bAuftrStartA:= TRUE;
			bAuftrStartB:= FALSE;
	ELSE
		bAuftrStartA:= FALSE;
		bAuftrStartB:= FALSE;
	END_IF

2: (*AchsStart "B"*)

	IF bAuftrStart
		THEN
			bAuftrStartA:= FALSE;
			bAuftrStartB:= TRUE;
	ELSE
		bAuftrStartA:= FALSE;
		bAuftrStartB:= FALSE;
	END_IF

	END_CASE

	// Achs-Fahrauftrag stoppen
	bAuftrStop	:= IQ_stAchse.stAuftrg.bPTP_stop
						OR (IQ_stAchse.stAuftrg.bPTP_AutoStop
							AND I_bAutoStopAktiv);

	// Achs-Fahrauftrag verzögern
	IF IQ_stAchse.stAuftrg.bPTP_verz
	THEN
		fAuftrOverride	:=
			MIN ( IQ_stAchse.stFreigb.fOverride,	// Override über die Achsstruktur
			MIN ( I_fOverride,	// Override über den Eingang am Achs-Baustein
					fOverridePTP));	// maximaler Override über die globale Variable
	ELSE
		fAuftrOverride	:=
			MIN(I_fOverride,
			fOverridePTP);	// maximaler Override über die globale Variable
	END_IF

	// Achs-Fahrauftrag anhalten
	IF IQ_stAchse.stAuftrg.bPTP_halt
		THEN
			fAuftrOverride:= 0;	// Override 0%
	END_IF

	(*Achs-Fahrauftrag freigeben*)
	IF NOT bAuftrStart
		AND IQ_stAchse.bBetrbBer
		AND IQ_stAchse.stFreigb.bVorsFrgPos
		AND IQ_stAchse.stFreigb.bVorsFrgNeg
		THEN
			IQ_stAchse.stAuftrg.bPTP_PosiFrg:= TRUE;
		ELSE
			IQ_stAchse.stAuftrg.bPTP_PosiFrg:= FALSE;
	END_IF

	(*Achs-Fahrauftrag ausführen*)

	IF fAuftrZielPos >= 0 (*Richtungsvorgabe*)
		THEN
			fbAchsStartA2.Direction:=
			fbAchsStartB2.Direction:= MC_Positive_Direction;
		ELSE
			fbAchsStartA2.Direction:=
			fbAchsStartB2.Direction:= MC_Negative_Direction;
	END_IF

	fbAchsStartA2 (Axis				:= IQ_fbAxisRef,
				      Execute			:= bAuftrStartA,
				      Velocity			:= fAuftrGeschw,
				      Acceleration	:= 0,	(*SystemManager*)
				      Deceleration	:= 0,	(*SystemManager*)
				      Jerk				:= 0,	(*SystemManager*)
				      BufferMode		:= nAuftrBuffMode,

					   Active			=> bAuftrAktivA,
				      InVelocity		=> ,

				      Busy				=>	stAchsStartAOut.Busy,
				      Error				=>	stAchsStartAOut.Error,
				      ErrorID			=>	stAchsStartAOut.ErrorID);

	fbAchsStartB2 (Axis				:= IQ_fbAxisRef,
				      Execute			:= bAuftrStartB,
				      Velocity			:= fAuftrGeschw,
				      Acceleration	:= 0,	(*SystemManager*)
				      Deceleration	:= 0,	(*SystemManager*)
				      Jerk				:= 0,	(*SystemManager*)
				      BufferMode		:= nAuftrBuffMode,

					   Active			=> bAuftrAktivB,
				      InVelocity		=> ,

				      Busy				=>	stAchsStartBOut.Busy,
				      Error				=>	stAchsStartBOut.Error,
				      ErrorID			=>	stAchsStartBOut.ErrorID);

	fbAchsStop    (Axis				:= IQ_fbAxisRef,
				      Execute			:= bAuftrStop,
				      Deceleration	:= 0,	(*SystemManager*)
				      Jerk				:= 0,	(*SystemManager*)
				      BufferMode		:= MC_Aborting,

				      Done				=> bAuftrGestoppt,

				      Busy				=>	stAchsStopOut.Busy,
				      Error				=>	stAchsStopOut.Error,
				      ErrorID			=>	stAchsStopOut.ErrorID);


	IQ_stAchse.stAuftrg.fPTP_LetzZiel:= 0;

	IQ_stAchse.stAuftrg.bPTP_aktiv	:= (bAuftrStartA AND bAuftrAktivA)
										   		 				OR (bAuftrStartB AND bAuftrAktivB);
	IQ_stAchse.stAuftrg.bPTP_inZiel	:= FALSE;
	IQ_stAchse.stAuftrg.bPTP_inFenst	:= FALSE;
	IQ_stAchse.stAuftrg.bPTP_gest		:= bAuftrGestoppt;

	(*Laufzeitmeldung Fahrauftrag*)

	IQ_stAchse.stMeldg.bLfZeitFehl:= FALSE;
END_ACTION

ACTION i_AchsModulo:
	(*Achswerte schreiben / Achse starten / Achse stoppen*)
	(*-Endlosachse*)

	IQ_stAchse.stAuftrg.sPTP_AuftrgTyp:= 'Modulobetrieb';

	IF IQ_stAchse.stAuftrg.arrPTP_start[cKopplPos]		(*Korrekt-Koppelposition*)
		THEN
			fAuftrZielPos	:= IQ_stAchse.stKoppln.fKorrektPos;
			fAuftrGeschw	:= IQ_stAchse.stParam.fEilgGeschw * 0.05;
	ELSIF IQ_stAchse.stAuftrg.arrPTP_start[cGrundPos]	(*Grundstellungsposition*)
		THEN
			fAuftrZielPos	:= IQ_stAchse.stParam.fGrdstlgPos;
			fAuftrGeschw	:= IQ_stAchse.stParam.fEilgGeschw * 0.25;
	ELSIF IQ_stAchse.stAuftrg.arrPTP_start[cBearbPos]	(*Bearbeitungsposition*)
		THEN
			fAuftrZielPos	:= IQ_stAchse.stAuftrg.fPTP_ZielPos
									+ IQ_stAchse.stParam.fPosVerrWert
									+ IQ_stAchse.stParam.fPosOffsWert;
			fAuftrGeschw	:= (IQ_stAchse.stParam.fEilgGeschw / 100)
   								 * IQ_stAchse.stAuftrg.fPTP_Geschw;
	END_IF

	(*Achs-Fahrauftrag prüfen/starten*)

	IF IQ_stAchse.stAuftrg.arrPTP_start[cKopplPos]
		OR IQ_stAchse.stAuftrg.arrPTP_start[cGrundPos]
		OR IQ_stAchse.stAuftrg.arrPTP_start[cBearbPos]
		THEN
			IF (IQ_stAchse.stParam.bSoftEndlAkt
				AND fAuftrZielPos >= IQ_stAchse.stParam.fSoftEndlMin
				AND fAuftrZielPos <= IQ_stAchse.stParam.fSoftEndlMax)
				OR IQ_stAchse.stParam.bOhnSoftEndl
				THEN
					IF NOT bAuftrStart
						OR bNeuAuftrVorg
						THEN
							IF NOT bAuftrStart
								THEN
									nAuftrBuffMode:= IQ_stAchse.stAuftrg.ePTP_BuffMode;
								ELSE
									nAuftrBuffMode:= MC_Aborting;
							END_IF

							IF NOT bAuftrStop
							THEN
								bAuftrStart:= TRUE;
							END_IF

							IF nAuftrState = 1
								THEN
									nAuftrState:= 2;
								ELSE
									nAuftrState:= 1;
							END_IF

							bNeuAuftrVorg:= FALSE;

							fLetztZielPos:= fAuftrZielPos;
							fLetztGeschw:= fAuftrGeschw;
						ELSE
							bNeuAuftrVorg:= (fAuftrZielPos <> fLetztZielPos
											 	 		OR fAuftrGeschw <> fLetztGeschw)
													AND NOT bAuftrStop;
					END_IF
				ELSE
					bAuftrStart:= FALSE;
					bNeuAuftrVorg:= FALSE;
					IQ_stAchse.stMeldg.bZielPosFehl:= TRUE;
			END_IF
		ELSE
			bAuftrStart:= FALSE;
			bNeuAuftrVorg:= FALSE;
			IQ_stAchse.stMeldg.bZielPosFehl:= FALSE;
	END_IF

	CASE nAuftrState OF

1: (*AchsStart "A"*)

	IF bAuftrStart
		THEN
			bAuftrStartA:= TRUE;
			bAuftrStartB:= FALSE;
	ELSE
		bAuftrStartA:= FALSE;
		bAuftrStartB:= FALSE;
	END_IF

2: (*AchsStart "B"*)

	IF bAuftrStart
		THEN
			bAuftrStartA:= FALSE;
			bAuftrStartB:= TRUE;
	ELSE
		bAuftrStartA:= FALSE;
		bAuftrStartB:= FALSE;
	END_IF

	END_CASE

	// Achs-Fahrauftrag stoppen
	bAuftrStop	:= IQ_stAchse.stAuftrg.bPTP_stop
						OR (IQ_stAchse.stAuftrg.bPTP_AutoStop
							AND I_bAutoStopAktiv);

	// Achs-Fahrauftrag verzögern
	IF IQ_stAchse.stAuftrg.bPTP_verz
	THEN
		fAuftrOverride	:=
			MIN ( IQ_stAchse.stFreigb.fOverride,	// Override über die Achsstruktur
			MIN ( I_fOverride,	// Override über den Eingang am Achs-Baustein
					fOverridePTP));	// maximaler Override über die globale Variable
	ELSE
		fAuftrOverride	:=
			MIN(I_fOverride,
			fOverridePTP);	// maximaler Override über die globale Variable
	END_IF

	// Achs-Fahrauftrag anhalten
	IF IQ_stAchse.stAuftrg.bPTP_halt
		THEN
			fAuftrOverride:= 0;	// Override 0%
	END_IF

	(*Achs-Fahrauftrag freigeben*)
	IF NOT bAuftrStart
		AND IQ_stAchse.bBetrbBer
		AND IQ_stAchse.stFreigb.bVorsFrgPos
		AND IQ_stAchse.stFreigb.bVorsFrgNeg
		THEN
			IQ_stAchse.stAuftrg.bPTP_PosiFrg:= TRUE;
		ELSE
			IQ_stAchse.stAuftrg.bPTP_PosiFrg:= FALSE;
	END_IF

	(*Achs-Fahrauftrag ausführen*)
	fbAchsStartA3 (Axis				:= IQ_fbAxisRef,
				      Execute			:= bAuftrStartA,
				      Velocity			:= fAuftrGeschw,
				      Position			:= fAuftrZielPos,
				      Acceleration	:= 0,	(*SystemManager*)
				      Deceleration	:= 0,	(*SystemManager*)
				      Jerk				:= 0,	(*SystemManager*)
				      BufferMode		:= nAuftrBuffMode,
						Direction		:= I_eRichtungModulo,

					   Active			=> bAuftrAktivA,
				      Done				=> bAuftrFertigA,

				      Busy				=>	stAchsStartAOut.Busy,
				      Error				=>	stAchsStartAOut.Error,
				      ErrorID			=>	stAchsStartAOut.ErrorID);

	fbAchsStartB3 (Axis				:= IQ_fbAxisRef,
				      Execute			:= bAuftrStartB,
				      Velocity			:= fAuftrGeschw,
				      Position			:= fAuftrZielPos,
				      Acceleration	:= 0,	(*SystemManager*)
				      Deceleration	:= 0,	(*SystemManager*)
				      Jerk				:= 0,	(*SystemManager*)
				      BufferMode		:= nAuftrBuffMode,
						Direction		:= I_eRichtungModulo,

					   Active			=> bAuftrAktivB,
				      Done				=> bAuftrFertigB,

				      Busy				=>	stAchsStartBOut.Busy,
				      Error				=>	stAchsStartBOut.Error,
				      ErrorID			=>	stAchsStartBOut.ErrorID);

	fbAchsStop    (Axis				:= IQ_fbAxisRef,
				      Execute			:= bAuftrStop,
				      Deceleration	:= 0,	(*SystemManager*)
				      Jerk				:= 0,	(*SystemManager*)
				      BufferMode		:= MC_Aborting,

				      Done				=> bAuftrGestoppt,

				      Busy				=>	stAchsStopOut.Busy,
				      Error				=>	stAchsStopOut.Error,
				      ErrorID			=>	stAchsStopOut.ErrorID);



	IQ_stAchse.stAuftrg.fPTP_LetzZiel:= fLetztZielPos;
	
	IQ_stAchse.stAuftrg.bPTP_aktiv	:= (bAuftrStartA AND bAuftrAktivA)
										   		 		 		OR (bAuftrStartB AND bAuftrAktivB);
	IQ_stAchse.stAuftrg.bPTP_inZiel	:= (bAuftrStartA AND bAuftrFertigA)
										    		  		  		OR (bAuftrStartB AND bAuftrFertigB);
	IQ_stAchse.stAuftrg.bPTP_inFenst	:= IQ_stAchse.fPosIstwert < (fLetztZielPos + 0.1)
													  		  		AND IQ_stAchse.fPosIstwert > (fLetztZielPos - 0.1);
	IQ_stAchse.stAuftrg.bPTP_gest		:= bAuftrGestoppt;
	
	(*Laufzeitmeldung Fahrauftrag*)

	tonAuftrLfZeit (IN:= bAuftrStart
							   AND NOT IQ_stAchse.stAuftrg.bPTP_stop
						      AND NOT IQ_stAchse.stAuftrg.bPTP_halt
						      AND NOT IQ_stAchse.stAuftrg.bPTP_inZiel,
					    PT:= T#60S);

	IQ_stAchse.stMeldg.bLfZeitFehl:= tonAuftrLfZeit.Q;
END_ACTION

ACTION k_AchsReset:
	(*Achse zurücksetzen*)

	fbAchsReset (Axis				:= IQ_fbAxisRef,
				    Execute			:= IQ_stAchse.stGrdfkt.bReset_ausf,

				    Busy				=>	stAchsResetOut.Busy,
				    Error			=>	stAchsResetOut.Error,
				    ErrorID			=>	stAchsResetOut.ErrorID);
					 
	tpReset(	IN:= NOT bInit
						OR bFehlerEtherCATAllg,
				PT:= t#10s);

	bInit := TRUE;
	
	IQ_stAchse.stEinAusG.Q_nSignalsteuerwort.0 := ((IQ_stAchse.bNcFehler
																					OR NOT IQ_stAchse.bBetrbBer)
																					AND IQ_stAchse.stGrdfkt.bReset_ausf)
																					OR tpReset.Q ;
END_ACTION

ACTION x_AchsMeldg:
	(*Achsmeldungen ausgeben*)

	//Meldeausgabe s."FB_UniAchsAnstg"
END_ACTION

END_FUNCTION_BLOCK

// POUs/FB_AchsStartAusf
FUNCTION_BLOCK FB_AchsStartAusf
VAR_IN_OUT
	IQ_stAchse			:TC3_UniLib.ST_NcAchsen;	// Schnittstelle zur NC-Achse
END_VAR
VAR_INPUT

	I_nSchutzBer		:INT;	// Schutzbereichs-ID für Abfrage Automatik ein und Steuerung ein

	I_bAchse_zurGrdP	:BOOL;	// arrPTP_start[cGrundPos] wird angestoßen
	I_bAchse_zurArbP	:BOOL;	// arrPTP_start[cBearbPos] wird angestoßen
	I_bAchse_stopPos	:BOOL;	// Achs wird über bPTP_stop gestoppt

	I_bAchse_FrgGrdP	:BOOL;	// Freigabe zur Grundposition zu fahren
	I_bAchse_FrgArbP	:BOOL;	// Freigabe zur Bearbeitungsposition zu fahren
	I_bAchse_FrgRglP	:BOOL;	// Freigabe die Zielposition zu halten/ bzw. nochmal anzufahren, wenn Zielposition +-2 der Istpos entspricht.

	(*ToDo: AchsEinzlStart
			  AchsNachStart
			  AchsNachRegeln
			  AchsOverride	
			  AchsStopp*)

END_VAR
VAR_OUTPUT
	Q_bAchsePosFehl	:BOOL;	// Bei I_bAchse_FrgRglP wenn die Istposition nicht innerhalb +-2 liegt, TRUE

	Q_bAchse_aktiv		:BOOL;	// Abbildung von bPTP_aktiv wenn ein Achsstart ansteht.
	Q_bAchse_inPos		:BOOL;	// Abbildung von bPTP_inZiel wenn ein Achsstart ansteht.
	Q_bAchse_gestPos	:BOOL;	// Abbildung von bPTP_gest wenn ein Achsstart ansteht.
END_VAR
VAR

	bAchse_zurRglP	:BOOL;
	bAchse_inRglP	:BOOL;

	bAchse_start	:BOOL;
	bAchse_stop		:BOOL;

	tonAntrFrg		:Tc2_Standard.TON;
	
	nStepAchsStop	:INT;

END_VAR


IF I_nSchutzBer <= 0
THEN RETURN;
END_IF

	(*Achs-Fahrauftrag ausführen*)

	IF NOT bAchse_inRglP
		AND IQ_stAchse.fPosIstwert < (IQ_stAchse.stAuftrg.fPTP_ZielPos + 2)
		AND IQ_stAchse.fPosIstwert > (IQ_stAchse.stAuftrg.fPTP_ZielPos - 2)
		AND arrBetrartAutomAktiv[I_nSchutzBer]
	THEN
		bAchse_zurRglP	:= TRUE;
	END_IF

	IF NOT I_bAchse_FrgRglP
		OR I_bAchse_zurGrdP
		OR I_bAchse_zurArbP
		OR (bAchse_zurRglP
		AND Q_bAchse_inPos)
	THEN
		bAchse_zurRglP	:= FALSE;
		bAchse_inRglP	:= TRUE;
	END_IF

	IF NOT IQ_stAchse.stFreigb.bReglerFrg
		THEN
			bAchse_inRglP:= FALSE;
	END_IF

	IF I_bAchse_FrgRglP
		AND (IQ_stAchse.fPosIstwert >= (IQ_stAchse.stAuftrg.fPTP_ZielPos + 2)
		OR IQ_stAchse.fPosIstwert <= (IQ_stAchse.stAuftrg.fPTP_ZielPos - 2))
		AND arrBetrartAutomAktiv[I_nSchutzBer]
			THEN
				Q_bAchsePosFehl:= TRUE;
			ELSE
				Q_bAchsePosFehl:= FALSE;
	END_IF

	(**********************************************************************)

	IF I_bAchse_zurGrdP
		OR I_bAchse_zurArbP
		OR bAchse_zurRglP
		THEN
			IF NOT Q_bAchse_inPos
				AND NOT Q_bAchse_gestPos
				AND (I_bAchse_FrgGrdP OR NOT I_bAchse_zurGrdP)
				AND (I_bAchse_FrgArbP OR NOT I_bAchse_zurArbP)
				AND IQ_stAchse.stAuftrg.bPTP_PosiFrg
				THEN
					bAchse_start:= TRUE;
			END_IF

			IF bAchse_start
				AND I_bAchse_stopPos
			THEN
				bAchse_stop:= TRUE;
			ELSIF NOT I_bAchse_stopPos
			THEN
				bAchse_stop:= FALSE;
			END_IF
			
			IF bAchse_start
				THEN
					IF IQ_stAchse.stAuftrg.bPTP_aktiv
						THEN
							Q_bAchse_aktiv:= TRUE;
					END_IF
					IF IQ_stAchse.stAuftrg.bPTP_inZiel
						THEN
							Q_bAchse_aktiv	 := FALSE;
							Q_bAchse_inPos	 := TRUE;
							bAchse_start	 := FALSE;
							bAchse_stop 	 := FALSE;
							nStepAchsStop	 := 0;
					END_IF
					IF IQ_stAchse.stAuftrg.bPTP_gest
						THEN
							Q_bAchse_aktiv	 := FALSE;
							Q_bAchse_gestPos:= TRUE;
							bAchse_start	 := FALSE;
							bAchse_stop 	 := FALSE;
					END_IF
			END_IF
		ELSE
			Q_bAchse_aktiv	 := FALSE;
			Q_bAchse_inPos	 := FALSE;
			Q_bAchse_gestPos:= FALSE;
			bAchse_start	 := FALSE;
			bAchse_stop 	 := FALSE;
	END_IF

	IF bAchse_start
		THEN
			IQ_stAchse.stAuftrg.bPTP_AutoStop	:= FALSE;
					
			IF I_bAchse_zurGrdP
				THEN
					IQ_stAchse.stAuftrg.arrPTP_start[cGrundPos]:= tonAntrFrg.Q;
					IQ_stAchse.stAuftrg.arrPTP_start[cBearbPos]:= FALSE;
			ELSIF I_bAchse_zurArbP
				OR bAchse_zurRglP
				THEN
					IQ_stAchse.stAuftrg.arrPTP_start[cGrundPos]:= FALSE;
					IQ_stAchse.stAuftrg.arrPTP_start[cBearbPos]:= tonAntrFrg.Q;
					nStepAchsStop	:= 1;
			END_IF
			IQ_stAchse.stAuftrg.bPTP_stop:= bAchse_stop;
		ELSE
			IQ_stAchse.stAuftrg.arrPTP_start[cGrundPos]:= FALSE;
			IQ_stAchse.stAuftrg.arrPTP_start[cBearbPos]:= FALSE;
			IQ_stAchse.stAuftrg.bPTP_stop:= FALSE;
			
			CASE nStepAchsStop OF
			 0: //keine Achsbewegung vorhanden
				 IQ_stAchse.stAuftrg.bPTP_AutoStop:= FALSE;
			
			 1: // Achsen Stoppen, wenn keine Automatik aktiv 
				IF NOT arrBetrartAutomAktiv[I_nSchutzBer]
				THEN
					IQ_stAchse.stAuftrg.bPTP_AutoStop	:= TRUE;
					nStepAchsStop	:= 2;
				END_IF
			 
			 2: // Achsen ist gestoppt 
				IF IQ_stAchse.stAuftrg.bPTP_gest
					OR arrBetrartAutomAktiv[I_nSchutzBer]	 
				THEN
					IQ_stAchse.stAuftrg.bPTP_AutoStop	:= FALSE;
    				nStepAchsStop	:= 0;
				END_IF
		END_CASE
	END_IF

	tonAntrFrg (IN:= arrAchsGruppeFrgVerz[I_nSchutzBer],
					  PT:= T#1500MS);

// ENDE

END_FUNCTION_BLOCK

// POUs/FB_Bremsentest_BremseEinschleifen
// Funktionsbaustein für den Bremsentest und das Einschleifen einer Bremse an einem Bosch-Servo
FUNCTION_BLOCK FB_Bremsentest_BremseEinschleifen
VAR CONSTANT
   cVorwarnungBremsentest              : UDINT := 930069 ;                        // entspricht E3115
   cUberschreitungZeitBremsentest      : UDINT := 2044181 ;                      // entspricht F3115
END_VAR
VAR_INPUT
	I_bStart										: BOOL;	// Start, Triggert den Bremsentest
	I_bAchsfreigabe							: BOOL;	// Achsfreigabe/Achse Betriebsbereit für Einschleifen und Bremsentest
	I_bReset										: BOOL;	// Reset Fehler
	I_bResetEinschleifen						: BOOL;	// Nur einen Fehler im Einschleifvorgang quittieren
	I_bFatalErrorQuitt						: BOOL;	// Reset fatalen Fehler
	I_bOhneNennmomentAbfr					: BOOL;	// Gehaltenes Nennmoment der Bremse wird nicht überprüft. Z.B. wenn das Haltemoment der Bremse höhe ist als das Maximalmoment des Servos
	
	I_nStatus									: WORD;	// Verknüfung zur Bosch-Rexroth-Achse
	I_nDiagNummer								: DWORD; // Verknüfung zur Bosch-Rexroth-Achse
	I_nBetriebsstunden						: UDINT;	// Verknüfung zur Bosch-Rexroth-Achse
	
	I_sDateipfad								: Tc2_System.T_MaxString; // Dateipfad für die Log Datei
	I_sDateiname								: Tc2_System.T_MaxString; // Dateipfad für die Log Datei
	
	//Eingänge Bremse manuell einschleifen
	I_bAchseInGrdstlg									: BOOL;							//Achse ist in Grundstellung, Bremse darf manuell eingeschliffen werden
	I_bBremseManuellEinschleifen					: BOOL;							//Startkommando, dass die Bremse eingeschliffen werden soll
	I_tZeitBremseGeschl								: TIME := T#400MS;			//Zeit, die die Bremse während der Fahrt geschlossen sein soll (Standardmäßig auf 400ms eingestellt --> Vorgabe Bosch)
	I_fVerfahrwegEinschleifvorgang				: LREAL := 2;					//Der Weg, der die Achse beim Einschleifen verfährt (Standardmäßig auf 2mm eingestellt)
	I_bEinschlPosRichtung							: BOOL;							//Einschleifen der Bremse soll in positiver Richtung erfolgen
	I_bEinschlNegRichtung							: BOOL;							//Einschleifen der Bremse soll in negativer Richtung erfolgen
	I_bDrehachse										: BOOL;							//Ist eine rotatorische und keine lineare Achse, dann wird I_fVorgabeGeschwEinschleifenRotatorisch gewählt
	I_fVorgabeGeschwEinschleifenLinear			: LREAL := 1.666666666;		//Geschwindigkeit mit der die Bremse eingeschliffen werden soll in mm/s
	I_fVorgabeGeschwEinschleifenRotatorisch	: LREAL;							//Geschwindigkeit mit der die Bremse eingeschliffen werden soll (rotatorische Achse) in °/s
	I_bHandbetriebAktiv								: BOOL;							//Bremse Einschleifen nur Starten, wenn Handbetrieb aktiv und Automatik aus
	I_bTakt												: BOOL;							//Takt für die Handfunktionsanzeige
	I_stZeitstempel									: TC3_UniLib.ST_TimeStruct;	//Zeitstempel zum Schreiben der Logdatei
END_VAR
VAR_OUTPUT
	Q_bStart							: BOOL;	// Signal Start Bremsentest an Achse
	Q_bDone							: BOOL;	// Signal Fertig an Ablauf
	
	Q_bVorwarnungZeitintervall	: BOOL;
	Q_bWarteAufNaechstenTest	: BOOL;
	Q_bErr_Haltebremse			: BOOL;	// Signal vom Servo: Haltebremse ist nicht OK.
	Q_bErr_Bremsoeffnung			: BOOL;	// Signal vom Servo: Bremsöffnung ist nicht OK
	Q_bErr_Haltemoment			: BOOL;	// Signal vom Servo: Gehaltenes Moment ist nicht OK
	Q_bErr_Ueberlast				: BOOL;	// Signal vom Servo: Last für Servo ist nicht OK
	Q_bErr_Drahtbruchtest		: BOOL;	// Signal vom Servo: Verdrahtung ist nicht OK.
	Q_bErr_Nennmoment				: BOOL;	// Signal vom Servo: Nennmoment ist nicht OK, wenn überwacht.
	Q_bError							: BOOL;	// Bremsentest nicht erfolgreich -> nächster Test in 15 min
	Q_bFatalError					: BOOL;	// Bremsentest 10x hintereinander nicht erfolgreich
	Q_sLogZeile						: Tc2_System.T_MaxString;
	Q_sError							: Tc2_System.T_MaxString;
	Q_bHaltebremse_OK				: BOOL;	// Signal vom Servo: Haltebremse ist OK.
	
	//Ausgänge Bremse manuell einschleifen
	Q_bAutomatikSperren			: BOOL;	//Automatik Einschalten sollte gesperrt werden, während des Einschleifvorgangs der Bremse
	Q_bBremseSchliessen			: BOOL;	//Bremse manuell schließen wenn die Antriebsfreigabe gesetzt ist (Kommando C3800 P-0-0543 auf das Steuerwort der Achse verknüpfen)
	Q_bBremseEinschleifenAktiv	: BOOL;	//Einschleifvorgang aktiv
	Q_nStatusHandfunktion		: BYTE;	//Status für die Darstellung der Handfuktionstasten in der Applikation
END_VAR
VAR_IN_OUT
	IQ_stUniAnstg					: ST_UniEinschleifen;	//Button für das Starten des Einschleifens der Achse	

	IQ_fbAchsStartAusfuehren	: FB_AchsStartAusf;			// Achse fürs Einschleifen starten
	IQ_stAchse						: TC3_UniLib.ST_NcAchsen;	// Schnittstelle zur Achse
END_VAR
VAR
	bSpannung24V					: BOOL;
	bHaltebremse_OK				: BOOL;
	bBremsoeffnung_OK				: BOOL;
	bHaltemoment_OK				: BOOL;
	bUeberlast_OK					: BOOL;
	bDrahtbruchtest_OK			: BOOL;
	bReserviert						: BOOL;
	bNennmoment_OK					: BOOL;
	bFehlerBremsentest			: BOOL;
	bOhneFehlerBremsentest		: BOOL;	// um bei erneutem Bremsentest bei einem fehlerhaftem Test, nicht wieder alle Tests der Achsen zu starten	

	sDiagString						: STRING;
	
	nStd								: UINT;
	nMin								: UINT;
	nSek								: UINT;
	
	fbLogToFile						: TC3_UniLib.FB_LogToFile;
	
	rtrigStart						: R_TRIG;
	bBremsentestNotwendig		: BOOL;
	bBremsentestAktiv				: BOOL;
	
	sUeberschrift					: Tc2_System.T_MaxString :='Timestamp;Betriebsstunden;Haltebremse;Bremsöffnung;Haltemoment;Überlast;Drahtbruchtest;Nennmoment;$R';
	
	nState							: INT;
	nStateOld						: INT;
	tonTimeOver						: Tc2_Standard.TON;
	tonNeustart						: Tc2_Standard.TON;
	tonQuittOhneFehler			: Tc2_Standard.TON;
	nDauerSeitLetztemTest		: UDINT;
	
	//Manueller Einschleifvorgang der Bremse
	rTrigBremseEinschleifen		: Tc2_Standard.R_TRIG;
	rTrigResetEinschleifen		: Tc2_Standard.R_TRIG;
	tonBremseGeschl				: Tc2_Standard.TON;
	fPosIstwert						: LREAL;
	bBremseSchliessen				: BOOL;
	
	//Relevante Variablen zur Diagnose
	stUniAnstgFkt					:ST_UniBaustein;
END_VAR

VAR PERSISTENT
	nFehlerZaehler					: INT;
	nLetzterTest					: UDINT;
END_VAR


//*********************************************************************
a_LogZeile();
a_Error();
b_AnwEinschleifen();

//*********************************************************************
nStd := TO_UINT(I_nBetriebsstunden / 36000);
nMin := TO_UINT((I_nBetriebsstunden - (nStd * 36000)) / 600);
nSek := TO_UINT((I_nBetriebsstunden -(nStd * 36000) - (nMin* 600)) / 10);

//*********************************************************************
bSpannung24V					:=	I_nStatus.0;
bHaltebremse_OK				:=	I_nStatus.1;
bBremsoeffnung_OK				:=	I_nStatus.2;
bHaltemoment_OK				:=	I_nStatus.3;
bUeberlast_OK					:=	I_nStatus.4;
bDrahtbruchtest_OK			:=	I_nStatus.5;
bReserviert						:=	I_nStatus.6;
bNennmoment_OK					:=	I_nStatus.7;

Q_bHaltebremse_OK := bHaltebremse_OK;
//*********************************************************************

nDauerSeitLetztemTest := I_nBetriebsstunden 
								 	- nLetzterTest;

IF (nDauerSeitLetztemTest 
		> 279000) //Entspricht 8h
	OR (nLetzterTest
		> I_nBetriebsstunden)
	OR I_nStatus.8
THEN
	bBremsentestNotwendig := TRUE;
ELSIF bSpannung24V
	AND bHaltebremse_OK
	AND bBremsoeffnung_OK 	
	AND bHaltemoment_OK
	AND bUeberlast_OK
	AND bDrahtbruchtest_OK
	AND (bNennmoment_OK
		OR I_bOhneNennmomentAbfr)
THEN	
	Q_bErr_Haltebremse	:=	FALSE;
	Q_bErr_Bremsoeffnung	:=	FALSE;
	Q_bErr_Haltemoment	:=	FALSE;
	Q_bErr_Ueberlast		:=	FALSE;
	Q_bErr_Drahtbruchtest:=	FALSE;
	Q_bErr_Nennmoment		:=	FALSE;
	bFehlerBremsentest	:= FALSE;
	nFehlerZaehler			:= 0;
END_IF
// Nach Zeit wieder löschen, dann sind alle anderen fehlerhaften Achsen neu getestet worden
tonQuittOhneFehler(
	IN:= bOhneFehlerBremsentest,
	pt:= T#10M);
IF tonQuittOhneFehler.Q THEN	
	bOhneFehlerBremsentest:= FALSE;
END_IF
(***)
rtrigStart(
	Clk	:=	I_bStart
				AND NOT I_bReset
				AND NOT bOhneFehlerBremsentest);

rTrigResetEinschleifen(
	CLK := I_bResetEinschleifen
				AND nState >= 200
				AND nState <= 260
);

IF rTrigResetEinschleifen.Q
THEN
	IQ_fbAchsStartAusfuehren.I_bAchse_zurArbP := FALSE;
	nState := 0;
END_IF

//*********************************************************************

CASE nState OF
//////////////////////////////////////////////////////////////////////////	 
0:	// INIT
	Q_bStart 						:= 
	Q_bDone							:= 
	Q_bBremseEinschleifenAktiv :=
	Q_bAutomatikSperren			:=
	bBremsentestAktiv				:=
	bBremseSchliessen 			:= FALSE;
	
	IF (rtrigStart.Q
		AND NOT bOhneFehlerBremsentest)
		OR (bFehlerBremsentest
				AND NOT Q_bBremseEinschleifenAktiv)
	THEN	
		tonNeustart(IN:=FALSE);
		fbLogToFile(I_bStart := FALSE);
		nLetzterTest			:=	I_nBetriebsstunden;
		Q_bErr_Haltebremse	:=	FALSE;
		Q_bErr_Bremsoeffnung	:=	FALSE;
		Q_bErr_Haltemoment	:=	FALSE;
		Q_bErr_Ueberlast		:=	FALSE;
		Q_bErr_Drahtbruchtest:=	FALSE;
		Q_bErr_Nennmoment		:=	FALSE;
		bOhneFehlerBremsentest	:= FALSE;
		nState					:=	5;
		
	//Sonderablauf, Bremse manuell einschleifen
	ELSIF rTrigBremseEinschleifen.Q
	THEN
		nState := 200;
	END_IF
//////////////////////////////////////////////////////////////////////////		
5: 
	bBremsentestAktiv := TRUE;

	IF I_bAchsfreigabe
	THEN
		nState					:=	10;
	END_IF
//////////////////////////////////////////////////////////////////////////		
10:	// Starte Bremsentest 
	Q_bStart 	:= TRUE;
	
	IF NOT bHaltebremse_OK
//		OR bFehlerBremsentest
	THEN
		nState	:=	20;
		bFehlerBremsentest := FALSE;
	ELSIF NOT I_bStart
		AND NOT bFehlerBremsentest
	THEN
		nState	:=	0;
	END_IF
	
//////////////////////////////////////////////////////////////////////////	
20:// Abfrage Ergebnisse
	tonTimeOver.PT := T#3S;
	
	IF bHaltebremse_OK
		AND bBremsoeffnung_OK	
		AND bHaltemoment_OK
		AND bUeberlast_OK
		AND bDrahtbruchtest_OK
		AND (bNennmoment_OK
			OR I_bOhneNennmomentAbfr)
	THEN
		Q_bStart					:= FALSE;
		bOhneFehlerBremsentest	:= TRUE;
		nFehlerZaehler			:= 0;
		nState					:=	30;
		
	ELSIF tonTimeOver.Q
	THEN
		Q_bStart					:= FALSE;
		Q_bErr_Haltebremse	:=	NOT bHaltebremse_OK;
		Q_bErr_Bremsoeffnung	:=	NOT bBremsoeffnung_OK;
		Q_bErr_Haltemoment	:=	NOT bHaltemoment_OK;
		Q_bErr_Ueberlast		:=	NOT bUeberlast_OK;
		Q_bErr_Drahtbruchtest:=	NOT bDrahtbruchtest_OK;
		Q_bErr_Nennmoment		:=	
			NOT bNennmoment_OK
			AND NOT I_bOhneNennmomentAbfr;
		bFehlerBremsentest	:= TRUE;
		nFehlerZaehler 		:= nFehlerZaehler + 1;
		nState					:=	30;
	END_IF

//////////////////////////////////////////////////////////////////////////	
30: // Speichern der Ergebnisse im File
	fbLogToFile(
		I_bStart				:= TRUE, 
		I_sDateipfad		:= I_sDateipfad, 
		I_sDateiname		:= I_sDateiname, 
		I_sUeberschrift	:= sUeberschrift,
		I_sZeile				:= Q_sLogZeile, 
		Q_bDone				=> );
	IF fbLogToFile.Q_bDone
	THEN
		nState					:=	100;
	END_IF
	
//////////////////////////////////////////////////////////////////////////	
100: // Auswertung, ob Fehler vorhanden sind
	bBremsentestAktiv := FALSE;
	
	IF rTrigBremseEinschleifen.Q
	THEN
		nState := 200;
	END_IF

	IF (nFehlerZaehler < 3)
		AND (nFehlerZaehler >= 2)
		AND (I_bReset
			OR rtrigStart.Q)
		AND NOT Q_bFatalError
	THEN
		nState  := 999;
	ELSIF (nFehlerZaehler > 0)	// 3 mal automatisch wiederholen, im Fehlerfall
			AND (nFehlerZaehler < 2) 	
			AND (I_bReset
				OR bFehlerBremsentest)
	THEN
		nState  := 999;
	ELSIF (nFehlerZaehler = 0)
	THEN
		nState  := 999;
	ELSIF (nFehlerZaehler
			>= 3) 
	THEN
		Q_bFatalError := TRUE;
		IF I_bFatalErrorQuitt
		THEN
			Q_bFatalError 	:= FALSE;
			nState  			:= 999;
			nFehlerZaehler	:= 0;
		END_IF
	END_IF

//////////////////////////////////////////////////////////////////////////	
999:	// Kontrolle ob Start Signal zurück genommen ist
	Q_bDone						:= TRUE;
	bBremsentestAktiv			:= FALSE;
	IF NOT bFehlerBremsentest THEN
		bBremsentestNotwendig 	:= FALSE;
	END_IF
	
	tonNeustart(	IN:= NOT I_bStart
								OR bFehlerBremsentest	,
						PT:= T#5S );
	IF tonNeustart.Q	
	THEN	 
		nState  := 0;
	END_IF
	
//////////////////////////////////////////////////////////////////////////	
200:	//Sonderablauf, Bremse manuell einschleifen

	Q_bAutomatikSperren 							:= 
	Q_bBremseEinschleifenAktiv					:= TRUE;
	fPosIstwert 									:= IQ_stAchse.fPosIstwert;

	nState := 210;
	
210:	//Geschwinigkeits- und Positionsvorgabe

	IF I_bDrehachse
	THEN
		IQ_stAchse.stAuftrg.fPTP_Geschw 			:= ((ABS(I_fVorgabeGeschwEinschleifenRotatorisch)
																	/ IQ_stAchse.stParam.fEilgGeschw)
																* 100);
	ELSE
		IQ_stAchse.stAuftrg.fPTP_Geschw 			:= ((ABS(I_fVorgabeGeschwEinschleifenLinear)
																	/ IQ_stAchse.stParam.fEilgGeschw)
																* 100);
	END_IF
																
	IQ_stAchse.stAuftrg.ePTP_BuffMode		:= MC_Aborting;
	
	//Auswahl der Richtung beim Einschleifen
	IF I_bEinschlNegRichtung
	THEN
		IQ_stAchse.stAuftrg.fPTP_ZielPos 	:= fPosIstwert - I_fVerfahrwegEinschleifvorgang;
		nState := 220;
	ELSIF I_bEinschlPosRichtung
	THEN
		IQ_stAchse.stAuftrg.fPTP_ZielPos 	:= fPosIstwert + I_fVerfahrwegEinschleifvorgang;
		nState := 220;
	END_IF
	
	
220:	//Achsauftrag starten und auf das Erreichen der Sollgeschwindigkeit warten
	
	IQ_fbAchsStartAusfuehren.I_bAchse_zurArbP := TRUE;
	
	//Überprüfen ob die Geschwindigkeit erreicht wird
	IF (ABS(IQ_stAchse.fVeloIstwert) >= I_fVorgabeGeschwEinschleifenRotatorisch)
		AND I_bDrehachse
	THEN
		tonBremseGeschl(IN := TRUE, PT := I_tZeitBremseGeschl);
		bBremseSchliessen := TRUE;
		nState := 230;
	ELSIF (ABS(IQ_stAchse.fVeloIstwert) >= I_fVorgabeGeschwEinschleifenLinear)
		AND NOT I_bDrehachse
	THEN
		tonBremseGeschl(IN := TRUE, PT := I_tZeitBremseGeschl);
		bBremseSchliessen := TRUE;
		nState := 230;
	END_IF
	
230:	//Zeit Bremse geschlossen abwarten

	tonBremseGeschl();
	
	//Warten bis die Bremse 400ms lang geschlossen war
	IF tonBremseGeschl.Q
	THEN
		tonBremseGeschl(IN := FALSE);
		bBremseSchliessen 		:= FALSE;
		nState 						:= 240;
	END_IF
	
240:	//Warten auf Achse in Position
	
	//Achse fährt weiter zur Positionsvorgabe
	IF IQ_fbAchsStartAusfuehren.Q_bAchse_inPos
	THEN
		IQ_fbAchsStartAusfuehren.I_bAchse_zurArbP := FALSE;
		nState 						:= 250; 
	END_IF
	
250:	//Achse auf vorherige Position fahren

	IQ_stAchse.stAuftrg.fPTP_ZielPos			:= fPosIstwert;
	IQ_stAchse.stAuftrg.fPTP_Geschw 			:= IQ_stAchse.stParam.fGeschwVorg;
	IQ_stAchse.stAuftrg.ePTP_BuffMode		:= MC_Aborting;
	
	nState := 260;
	
260:	//Achse auf vorherige Position fahren

	IQ_fbAchsStartAusfuehren.I_bAchse_zurArbP := TRUE;
	
	IF IQ_fbAchsStartAusfuehren.Q_bAchse_inPos
	THEN
		IQ_fbAchsStartAusfuehren.I_bAchse_zurArbP := FALSE;
		Q_bBremseEinschleifenAktiv						:= FALSE;
		Q_bAutomatikSperren 								:= FALSE;
		nState := 0;
	END_IF

END_CASE



//*********************************************************************
tonTimeOver(
	In:= nStateOld = nState);

nStateOld := nState;

//*********************************************************************
Q_bError := 
	Q_bErr_Haltebremse
	OR Q_bErr_Bremsoeffnung
	OR Q_bErr_Haltemoment
	OR Q_bErr_Ueberlast
	OR Q_bErr_Drahtbruchtest
	OR Q_bErr_Nennmoment
	OR bBremsentestNotwendig
	OR (TO_UDINT(I_nDiagNummer) = cUberschreitungZeitBremsentest);
	
Q_bVorwarnungZeitintervall :=
	bBremsentestNotwendig; // 15 min vor Ablauf der Zeit
							
Q_bBremseSchliessen := bBremseSchliessen
								AND I_bAchsfreigabe;

ACTION a_Error:
Q_sError := '';

IF Q_bVorwarnungZeitintervall
THEN
	Q_sError := 'Bremsentest innerhalb der nächsten 15min nötig!';
END_IF

IF TO_UDINT(I_nDiagNummer) = cUberschreitungZeitBremsentest
THEN
	Q_sError := 'Bremsentest nötig! Fehler quittieren und Bremsentest ausführen';
END_IF

IF Q_bErr_Bremsoeffnung
	OR Q_bErr_Haltebremse
	OR Q_bErr_Haltemoment
	OR Q_bErr_Ueberlast
	OR Q_bErr_Drahtbruchtest
	OR Q_bErr_Nennmoment
THEN
	Q_sError := 'Fehler beim Bremsentest';
END_IF

IF Q_bErr_Bremsoeffnung
THEN
	Q_sError := CONCAT(Q_sError,'| Fehler Bremsöffnung');
END_IF

IF Q_bErr_Haltebremse
THEN
	Q_sError := CONCAT(Q_sError,'| Fehler Haltebremse');
END_IF

IF Q_bErr_Haltemoment
THEN
	Q_sError := CONCAT(Q_sError,'| Fehler Haltemoment');
END_IF

IF Q_bErr_Ueberlast
THEN
	Q_sError := CONCAT(Q_sError,'| Fehler Überlast');
END_IF

IF Q_bErr_Drahtbruchtest
THEN
	Q_sError := CONCAT(Q_sError,'| Fehler Drahtbruchtest');
END_IF

IF Q_bErr_Nennmoment
THEN
	Q_sError := CONCAT(Q_sError,'| Fehler Nennmoment');
END_IF

IF nFehlerZaehler <> 0
THEN
	Q_sError := CONCAT(Q_sError,'-> ');
	Q_sError := CONCAT(Q_sError,TO_STRING(3-nFehlerZaehler));
	Q_sError := CONCAT(Q_sError,' Versuche übrig!');
END_IF

IF Q_bFatalError
THEN
	Q_sError := 'Schutzbereich stillgelegt -> Bremsfunktion defekt!';
END_IF
END_ACTION

ACTION a_LogZeile:

Q_sLogZeile := '';
Q_sLogZeile:= I_stZeitstempel.sTimeStamp;

IF Q_bErr_Haltebremse
THEN
	Q_sLogZeile:= CONCAT(Q_sLogZeile,'n.IO;');
ELSE
	Q_sLogZeile:= CONCAT(Q_sLogZeile,'IO;');
END_IF
IF Q_bErr_Bremsoeffnung
THEN
	Q_sLogZeile:= CONCAT(Q_sLogZeile,'n.IO;');
ELSE
	Q_sLogZeile:= CONCAT(Q_sLogZeile,'IO;');
END_IF
IF Q_bErr_Haltemoment
THEN
	Q_sLogZeile:= CONCAT(Q_sLogZeile,'n.IO;');
ELSE
	Q_sLogZeile:= CONCAT(Q_sLogZeile,'IO;');
END_IF
IF Q_bErr_Ueberlast
THEN
	Q_sLogZeile:= CONCAT(Q_sLogZeile,'n.IO;');
ELSE
	Q_sLogZeile:= CONCAT(Q_sLogZeile,'IO;');
END_IF
IF Q_bErr_Drahtbruchtest
THEN
	Q_sLogZeile:= CONCAT(Q_sLogZeile,'n.IO;');
ELSE
	Q_sLogZeile:= CONCAT(Q_sLogZeile,'IO;');
END_IF
IF Q_bErr_Nennmoment
THEN
	Q_sLogZeile:= CONCAT(Q_sLogZeile,'n.IO;');
ELSE
	Q_sLogZeile:= CONCAT(Q_sLogZeile,'IO;');
END_IF
END_ACTION

ACTION b_AnwEinschleifen:


stUniAnstgFkt.bHandAnw0 := IQ_stUniAnstg.stHandFktHMI[1].bySwitch > 0;

//Bremse manuell Einschleifen
rTrigBremseEinschleifen(
	CLK := stUniAnstgFkt.bHandAnw0
				AND I_bAchseInGrdstlg
				AND I_bHandbetriebAktiv
);

//Handfunktion Einschleifen
IF I_bHandbetriebAktiv
	AND NOT bBremsentestAktiv
	AND (I_bAchseInGrdstlg
			OR Q_bBremseEinschleifenAktiv)
THEN
	IF Q_bBremseEinschleifenAktiv
	THEN
		IF I_bTakt
		THEN
			stUniAnstgFkt.nHandStat := 1;
		ELSE
			stUniAnstgFkt.nHandStat := 0;
		END_IF
	ELSE
		stUniAnstgFkt.nHandStat := 0;
	END_IF
ELSE
	stUniAnstgFkt.nHandStat := 256;
END_IF

(*Zustände anzeigen*)

IF stUniAnstgFkt.nHandStat = 0		(*Funktion freigegeben*)
	THEN
		IQ_stUniAnstg.stHandFktHMI[1].sColour:= cDefaultAsString;
		IQ_stUniAnstg.stHandFktHMI[1].sText:= 'ausführen';
ELSIF stUniAnstgFkt.nHandStat = 1	(*Handfunktion aktiv*)
	THEN
		IQ_stUniAnstg.stHandFktHMI[1].sColour:= cGruenAsString;
		IQ_stUniAnstg.stHandFktHMI[1].sText:= 'ausführen';
ELSIF stUniAnstgFkt.nHandStat = 2	(*Handfunktion ausgeführt*)
	THEN
		IQ_stUniAnstg.stHandFktHMI[1].sColour:= cGruenAsString;
		IQ_stUniAnstg.stHandFktHMI[1].sText:= 'ausgeführt';
END_IF
IF stUniAnstgFkt.nHandStat = 256		(*Funktion gesperrt*)
	THEN
		IQ_stUniAnstg.stHandFktHMI[1].sColour	:= cDefaultAsString;
		IQ_stUniAnstg.stHandFktHMI[1].sText		:= 'ausführen';
		IQ_stUniAnstg.stHandFktHMI[1].byStatus	:= 1;
	ELSE
		IQ_stUniAnstg.stHandFktHMI[1].byStatus:= 0;
END_IF
END_ACTION

END_FUNCTION_BLOCK

// POUs/FB_BremsentestMitLog
// Bremsentest-Baustein für Bosch-Servos mit der neuen Firmware 
FUNCTION_BLOCK FB_BremsentestMitLog
VAR CONSTANT
	cVorwarnungBremsentest				: UDINT := 930069 ;		// entspricht E3115
	cUberschreitungZeitBremsentest	: UDINT := 2044181 ;		// entspricht F3115
END_VAR
VAR_INPUT
	I_bStart										: BOOL;	// Start 
	I_bAchsfreigabe							: BOOL;
	I_bReset										: BOOL;	// Reset Fehler
	I_bFatalErrorQuitt						: BOOL;	// Reset Fehler
	I_bOhneNennmomentAbfr					: BOOL;	// Nennmoment erreicht wird nicht abgefragt. Das ist wichtig, wenn ein Motor für die Bremse zu klein ausgewählt wurde. Dann erreicht der Motor das Nennmoment der Bremse nicht.
	
	I_nStatus									: WORD;	// Verknüfung zur Achse
	I_nDiagNummer								: DWORD; // Verknüfung zur Achse
	I_nBetriebsstunden						: UDINT;	// Verknüfung zur Achse
	
	I_sDateipfad								: Tc2_System.T_MaxString; // Dateipfad für die Log Datei
	I_sDateiname								: Tc2_System.T_MaxString; // Dateipfad für die Log Datei
	
	I_stZeitstempel							: TC3_UniLib.ST_TimeStruct;	//Zeitstempel zum Schreiben der Logdatei
END_VAR
VAR_OUTPUT
	Q_bStart							: BOOL;	// Signal an Achse
	Q_bDone							: BOOL;
	
	Q_bVorwarnungZeitintervall	: BOOL;
	Q_bWarteAufNaechstenTest	: BOOL;
	Q_bErr_Haltebremse			: BOOL;
	Q_bErr_Bremsoeffnung			: BOOL;
	Q_bErr_Haltemoment			: BOOL;
	Q_bErr_Ueberlast				: BOOL;
	Q_bErr_Drahtbruchtest		: BOOL;
	Q_bErr_Nennmoment				: BOOL;
	Q_bError							: BOOL;	// Bremsentest nicht erfolgreich -> nächster Test in 15 min
	Q_bFatalError					: BOOL;	// Bremsentest 10x hintereinander nicht erfolgreich
	Q_sLogZeile						: Tc2_System.T_MaxString;	
	Q_sError							: Tc2_System.T_MaxString;	
END_VAR
VAR
	bSpannung24V					: BOOL;
	bHaltebremse_OK				: BOOL;
	bBremsoeffnung_OK				: BOOL;
	bHaltemoment_OK				: BOOL;
	bUeberlast_OK					: BOOL;
	bDrahtbruchtest_OK			: BOOL;
	bReserviert						: BOOL;
	bNennmoment_OK					: BOOL;
	
	sDiagString						: STRING;
	
	nStd								: UINT;
	nMin								: UINT;
	nSek								: UINT;
	
	fbLogToFile						: TC3_UniLib.FB_LogToFile;
	
	rtrigStart						: Tc2_Standard.R_TRIG;
	bBremsentestNotwendig		: BOOL;
	
	sUeberschrift					: Tc2_System.T_MaxString :='Timestamp;Betriebsstunden;Haltebremse;Bremsöffnung;Haltemoment;Überlast;Drahtbruchtest;Nennmoment;$R';
	
	nState							: INT;
	nStateOld						: INT;
	tonTimeOver						: Tc2_Standard.TON;
	tonNeustart						: Tc2_Standard.TON;
END_VAR

VAR PERSISTENT
	nFehlerZaehler					: INT;
	nLetzterTest					: UDINT;
END_VAR

//*********************************************************************
a_LogZeile();
a_Error();
//*********************************************************************
nStd := LREAL_TO_UINT(I_nBetriebsstunden / 36000);
nMin := LREAL_TO_UINT((I_nBetriebsstunden - (nStd * 36000)) / 600);
nSek := LREAL_TO_UINT((I_nBetriebsstunden -(nStd * 36000) - (nMin* 600)) / 10);

//*********************************************************************
bSpannung24V					:=	I_nStatus.0;
bHaltebremse_OK				:=	I_nStatus.1;
bBremsoeffnung_OK				:=	I_nStatus.2;
bHaltemoment_OK				:=	I_nStatus.3;
bUeberlast_OK					:=	I_nStatus.4;
bDrahtbruchtest_OK			:=	I_nStatus.5;
bReserviert						:=	I_nStatus.6;
bNennmoment_OK					:=	I_nStatus.7;
//*********************************************************************
IF I_nStatus.8 // Bremsentest notwendig
THEN
	bBremsentestNotwendig := TRUE;
	
ELSIF bSpannung24V
	AND bHaltebremse_OK
	AND bBremsoeffnung_OK 	
	AND bHaltemoment_OK
	AND bUeberlast_OK
	AND bDrahtbruchtest_OK
	AND (bNennmoment_OK
		OR I_bOhneNennmomentAbfr)
THEN	// Wenn im Rexroth manuell ein Bremsentest ausgeführt wird und der fehlerfrei ist, dann werden hier die Fehler zurückgesetzt.
// Sonst würden die Fehler einfach anstehen bleiben, bis zum nächsten Bremsentest aus der SPS heraus.
	Q_bErr_Haltebremse	:=	FALSE;
	Q_bErr_Bremsoeffnung	:=	FALSE;
	Q_bErr_Haltemoment	:=	FALSE;
	Q_bErr_Ueberlast		:=	FALSE;
	Q_bErr_Drahtbruchtest:=	FALSE;
	Q_bErr_Nennmoment		:=	FALSE;
	nFehlerZaehler			:= 0;
END_IF

//*********************************************************************
rtrigStart(
	Clk	:=	I_bStart);
//*********************************************************************

CASE nState OF
//////////////////////////////////////////////////////////////////////////	 
0:	// INIT
	Q_bStart 	:= FALSE;
	Q_bDone		:= FALSE;
	IF rtrigStart.Q
	THEN
		tonNeustart(IN:=FALSE);
		fbLogToFile(I_bStart := FALSE);
		nLetzterTest			:=	I_nBetriebsstunden;
		Q_bErr_Haltebremse	:=	FALSE;
		Q_bErr_Bremsoeffnung	:=	FALSE;
		Q_bErr_Haltemoment	:=	FALSE;
		Q_bErr_Ueberlast		:=	FALSE;
		Q_bErr_Drahtbruchtest:=	FALSE;
		Q_bErr_Nennmoment		:=	FALSE;
		nState					:=	5;
	END_IF
//////////////////////////////////////////////////////////////////////////		
5: 
	IF I_bAchsfreigabe
	THEN
		nState					:=	10;
	END_IF
//////////////////////////////////////////////////////////////////////////		
10:	// Starte Bremsentest 
	Q_bStart 	:= TRUE;
	
	IF NOT bHaltebremse_OK
	THEN
		nState	:=	20;
	ELSIF NOT I_bStart
	THEN
		nState	:=	0;
	END_IF
	
//////////////////////////////////////////////////////////////////////////	
20:// Abfrage Ergebnisse
	tonTimeOver.PT := T#5S;
	
	IF bHaltebremse_OK
		AND bBremsoeffnung_OK	
		AND bHaltemoment_OK
		AND bUeberlast_OK
		AND bDrahtbruchtest_OK
		AND (bNennmoment_OK
			OR I_bOhneNennmomentAbfr)
	THEN
		Q_bStart					:= FALSE;
		nFehlerZaehler			:= 0;
		nState					:=	30;
		
	ELSIF tonTimeOver.Q
	THEN
		Q_bStart					:= FALSE;
		Q_bErr_Haltebremse	:=	NOT bHaltebremse_OK;
		Q_bErr_Bremsoeffnung	:=	NOT bBremsoeffnung_OK;
		Q_bErr_Haltemoment	:=	NOT bHaltemoment_OK;
		Q_bErr_Ueberlast		:=	NOT bUeberlast_OK;
		Q_bErr_Drahtbruchtest:=	NOT bDrahtbruchtest_OK;
		Q_bErr_Nennmoment		:=
			NOT bNennmoment_OK
			AND NOT I_bOhneNennmomentAbfr;
		
		nFehlerZaehler 		:= nFehlerZaehler + 1;
		nState					:=	30;
	END_IF

//////////////////////////////////////////////////////////////////////////	
30: // Speichern der Ergebnisse im File
	fbLogToFile(
		I_bStart				:= TRUE, 
		I_sDateipfad		:= I_sDateipfad, 
		I_sDateiname		:= I_sDateiname, 
		I_sUeberschrift	:= sUeberschrift,
		I_sZeile				:= Q_sLogZeile, 
		Q_bDone				=> );
	IF fbLogToFile.Q_bDone
	THEN
		nState					:=	100;
	END_IF
	
//////////////////////////////////////////////////////////////////////////	
100: // Auswertung, ob Fehler vorhanden sind
	IF (nFehlerZaehler < 3)
		AND (I_bReset
			OR rtrigStart.Q)
		AND NOT Q_bFatalError
	THEN
		nState  := 999;
	ELSIF (nFehlerZaehler = 0)
	THEN
		nState  := 999;
	ELSIF (nFehlerZaehler
			>= 3) 
	THEN
		Q_bFatalError := TRUE;
		IF I_bFatalErrorQuitt
		THEN
			Q_bFatalError 	:= FALSE;
			nState  			:= 999;
			nFehlerZaehler	:= 0;
		END_IF
	END_IF

//////////////////////////////////////////////////////////////////////////	
999:	// Kontrolle ob Start Signal zurück genommen ist
	Q_bDone						:= TRUE;
	bBremsentestNotwendig 	:= FALSE;
	tonNeustart(	IN:= NOT I_bStart,
						PT:= T#10S );
	IF tonNeustart.Q	
	THEN	 
		nState  := 0;
	END_IF

END_CASE

//*********************************************************************
tonTimeOver(
	In:= nStateOld = nState);

nStateOld := nState;

//*********************************************************************
Q_bError := 
	Q_bErr_Haltebremse
	OR Q_bErr_Bremsoeffnung
	OR Q_bErr_Haltemoment
	OR Q_bErr_Ueberlast
	OR Q_bErr_Drahtbruchtest
	OR Q_bErr_Nennmoment
	OR (TO_UDINT(I_nDiagNummer) = cUberschreitungZeitBremsentest);
	
Q_bVorwarnungZeitintervall :=
	bBremsentestNotwendig; // 15 min vor Ablauf der Zeit

ACTION a_Error:
Q_sError := '';

IF Q_bVorwarnungZeitintervall
THEN
	Q_sError := 'Bremsentest innerhalb der nächsten 15min nötig!';
END_IF

IF TO_UDINT(I_nDiagNummer) = cUberschreitungZeitBremsentest
THEN
	Q_sError := 'Bremsentest nötig! Fehler quittieren und Bremsentest ausführen';
END_IF

IF Q_bErr_Bremsoeffnung
	OR Q_bErr_Haltebremse
	OR Q_bErr_Haltemoment
	OR Q_bErr_Ueberlast
	OR Q_bErr_Drahtbruchtest
	OR Q_bErr_Nennmoment
THEN
	Q_sError := 'Fehler beim Bremsentest';
END_IF

IF Q_bErr_Bremsoeffnung
THEN
	Q_sError := CONCAT(Q_sError,'| Fehler Bremsöffnung');
END_IF

IF Q_bErr_Haltebremse
THEN
	Q_sError := CONCAT(Q_sError,'| Fehler Haltebremse');
END_IF

IF Q_bErr_Haltemoment
THEN
	Q_sError := CONCAT(Q_sError,'| Fehler Haltemoment');
END_IF

IF Q_bErr_Ueberlast
THEN
	Q_sError := CONCAT(Q_sError,'| Fehler Überlast');
END_IF

IF Q_bErr_Drahtbruchtest
THEN
	Q_sError := CONCAT(Q_sError,'| Fehler Drahtbruchtest');
END_IF

IF Q_bErr_Nennmoment
THEN
	Q_sError := CONCAT(Q_sError,'| Fehler Nennmoment');
END_IF

IF nFehlerZaehler <> 0
THEN
	Q_sError := CONCAT(Q_sError,'-> ');
	Q_sError := CONCAT(Q_sError,TO_STRING(10-nFehlerZaehler));
	Q_sError := CONCAT(Q_sError,' Versuche übrig!');
END_IF

IF Q_bFatalError
THEN
	Q_sError := 'Schutzbereich stillgelegt -> Bremsfunktion defekt!';
END_IF
END_ACTION

ACTION a_LogZeile:

Q_sLogZeile := '';
Q_sLogZeile:= I_stZeitstempel.sTimeStamp;

IF Q_bErr_Haltebremse
THEN
	Q_sLogZeile:= CONCAT(Q_sLogZeile,'n.IO;');
ELSE
	Q_sLogZeile:= CONCAT(Q_sLogZeile,'IO;');
END_IF
IF Q_bErr_Bremsoeffnung
THEN
	Q_sLogZeile:= CONCAT(Q_sLogZeile,'n.IO;');
ELSE
	Q_sLogZeile:= CONCAT(Q_sLogZeile,'IO;');
END_IF
IF Q_bErr_Haltemoment
THEN
	Q_sLogZeile:= CONCAT(Q_sLogZeile,'n.IO;');
ELSE
	Q_sLogZeile:= CONCAT(Q_sLogZeile,'IO;');
END_IF
IF Q_bErr_Ueberlast
THEN
	Q_sLogZeile:= CONCAT(Q_sLogZeile,'n.IO;');
ELSE
	Q_sLogZeile:= CONCAT(Q_sLogZeile,'IO;');
END_IF
IF Q_bErr_Drahtbruchtest
THEN
	Q_sLogZeile:= CONCAT(Q_sLogZeile,'n.IO;');
ELSE
	Q_sLogZeile:= CONCAT(Q_sLogZeile,'IO;');
END_IF
IF Q_bErr_Nennmoment
THEN
	Q_sLogZeile:= CONCAT(Q_sLogZeile,'n.IO;');
ELSE
	Q_sLogZeile:= CONCAT(Q_sLogZeile,'IO;');
END_IF
END_ACTION

END_FUNCTION_BLOCK

// POUs/FB_BremsentestMitLog_FW07
// Bremsentest-Baustein für Bosch-Servos mit der alten Firmware 
FUNCTION_BLOCK FB_BremsentestMitLog_FW07
VAR CONSTANT
	cVorwarnungBremsentest				: UDINT := 930069 ;		// entspricht E3115
	cUberschreitungZeitBremsentest	: UDINT := 995605 ;		// entspricht F3115
END_VAR
VAR_INPUT
	I_bStart										: BOOL;	// Start 
	I_bAchsfreigabe							: BOOL;
	I_bReset										: BOOL;	// Reset Fehler
	I_bFatalErrorQuitt						: BOOL;	// Reset Fehler
	
	I_nStatus									: WORD;	// Verknüfung zur Achse
	I_nDiagNummer								: DWORD; // Verknüfung zur Achse
	I_nBetriebsstunden						: UDINT;	// Verknüfung zur Achse
	
	I_sDateipfad								: Tc2_System.T_MaxString; // Dateipfad für die Log Datei
	I_sDateiname								: Tc2_System.T_MaxString; // Dateipfad für die Log Datei
	
	I_stZeitstempel							: TC3_UniLib.ST_TimeStruct;	//Zeitstempel zum Schreiben der Logdatei
END_VAR
VAR_OUTPUT
	Q_bStart							: BOOL;	// Signal an Achse
	Q_bDone							: BOOL;
	
	Q_bVorwarnungZeitintervall	: BOOL;
	Q_bErr_Haltebremse			: BOOL;
	Q_bErr_Bremsoeffnung			: BOOL;
	Q_bErr_Haltemoment			: BOOL;
	Q_bError							: BOOL;	// Bremsentest nicht erfolgreich -> nächster Test in 15 min
	Q_bFatalError					: BOOL;	// Bremsentest 10x hintereinander nicht erfolgreich
	Q_sLogZeile						: Tc2_System.T_MaxString;	
	Q_sError							: Tc2_System.T_MaxString;	
END_VAR
VAR
	bSpannung24V					: BOOL;
	bHaltebremse_OK				: BOOL;
	bBremsoeffnung_OK				: BOOL;
	bHaltemoment_OK				: BOOL;
	
	sDiagString						: STRING;
	
	nStd								: UINT;
	nMin								: UINT;
	nSek								: UINT;
	
	fbLogToFile						: TC3_UniLib.FB_LogToFile;
	
	rtrigStart						: Tc2_Standard.R_TRIG;
	bBremsentestNotwendig		: BOOL;
	
	sUeberschrift					: Tc2_System.T_MaxString :='Timestamp;Betriebsstunden;Haltebremse;Bremsöffnung;Haltemoment;$R';
	
	nState							: INT;
	nStateOld						: INT;
	tonTimeOver						: Tc2_Standard.TON;
	tonNeustart: Ton;
END_VAR

VAR PERSISTENT
	nFehlerZaehler					: INT;
	nLetzterTest					: UDINT;
END_VAR

//*********************************************************************
a_LogZeile();
a_Error();
//*********************************************************************
nStd := LREAL_TO_UINT(I_nBetriebsstunden / 36000);
nMin := LREAL_TO_UINT((I_nBetriebsstunden - (nStd * 36000)) / 600);
nSek := LREAL_TO_UINT((I_nBetriebsstunden -(nStd * 36000) - (nMin* 600)) / 10);

//*********************************************************************
bSpannung24V					:=	I_nStatus.0;
bHaltebremse_OK				:=	I_nStatus.1;
bBremsoeffnung_OK				:=	I_nStatus.2;
bHaltemoment_OK				:=	I_nStatus.3;
//*********************************************************************
IF TO_UDINT(I_nDiagNummer) = cVorwarnungBremsentest
THEN
	bBremsentestNotwendig := TRUE;
END_IF
//*********************************************************************
rtrigStart(
	Clk	:=	I_bStart);
//*********************************************************************

CASE nState OF
//////////////////////////////////////////////////////////////////////////	 
0:	// INIT
	Q_bStart 	:= FALSE;
	Q_bDone		:= FALSE;
	IF rtrigStart.Q
	THEN
		tonNeustart(IN:=FALSE);
		fbLogToFile(I_bStart := FALSE);
		nLetzterTest			:=	I_nBetriebsstunden;
		Q_bErr_Haltebremse	:=	FALSE;
		Q_bErr_Bremsoeffnung	:=	FALSE;
		Q_bErr_Haltemoment	:=	FALSE;
		nState					:=	5;
	END_IF
//////////////////////////////////////////////////////////////////////////		
5: 
	IF I_bAchsfreigabe
	THEN
		nState					:=	10;
	END_IF
//////////////////////////////////////////////////////////////////////////		
10:	// Starte Bremsentest 
	Q_bStart 	:= TRUE;
	
	IF NOT bHaltebremse_OK
	THEN
		nState	:=	20;
	ELSIF NOT I_bStart
	THEN
		nState	:=	0;
	END_IF
	
//////////////////////////////////////////////////////////////////////////	
20:// Abfrage Ergebnisse
	tonTimeOver.PT := T#5S;
	
	IF bHaltebremse_OK
		AND bBremsoeffnung_OK	
		AND bHaltemoment_OK
	THEN
		Q_bStart					:= FALSE;
		nFehlerZaehler			:= 0;
		nState					:=	30;
		
	ELSIF tonTimeOver.Q
	THEN
		Q_bStart					:= FALSE;
		Q_bErr_Haltebremse	:=	NOT bHaltebremse_OK;
		Q_bErr_Bremsoeffnung	:=	NOT bBremsoeffnung_OK;
		Q_bErr_Haltemoment	:=	NOT bHaltemoment_OK;
		
		nFehlerZaehler 		:= nFehlerZaehler + 1;
		nState					:=	30;
	END_IF

//////////////////////////////////////////////////////////////////////////	
30: // Speichern der Ergebnisse im File
	fbLogToFile(
		I_bStart				:= TRUE, 
		I_sDateipfad		:= I_sDateipfad, 
		I_sDateiname		:= I_sDateiname, 
		I_sUeberschrift	:= sUeberschrift,
		I_sZeile				:= Q_sLogZeile, 
		Q_bDone				=> );
	IF fbLogToFile.Q_bDone
	THEN
		nState					:=	100;
	END_IF
	
//////////////////////////////////////////////////////////////////////////	
100: // Auswertung, ob Fehler vorhanden sind
	IF (nFehlerZaehler
			< 10)
		AND I_bReset
	THEN
		nState  := 999;
	ELSIF (nFehlerZaehler = 0)
	THEN
		nState  := 999;
	ELSIF (nFehlerZaehler
			>= 10) 
	THEN
		Q_bFatalError := TRUE;
		IF I_bFatalErrorQuitt
		THEN
			Q_bFatalError 	:= FALSE;
			nState  			:= 999;
			nFehlerZaehler	:= 0;
		END_IF
	END_IF

//////////////////////////////////////////////////////////////////////////	
999:	// Kontrolle ob Start Signal zurück genommen ist
	Q_bDone						:= TRUE;
	bBremsentestNotwendig 	:= FALSE;
	tonNeustart(	IN:= NOT I_bStart,
						PT:= T#10S );
	IF tonNeustart.Q	
	THEN	 
		nState  := 0;
	END_IF

END_CASE

//*********************************************************************
tonTimeOver(
	In:= nStateOld = nState);

nStateOld := nState;

//*********************************************************************
Q_bError := 
	Q_bErr_Haltebremse
	OR Q_bErr_Bremsoeffnung
	OR Q_bErr_Haltemoment
	OR (TO_UDINT(I_nDiagNummer) = cUberschreitungZeitBremsentest);
	
Q_bVorwarnungZeitintervall :=
	bBremsentestNotwendig; // 15 min vor Ablauf der Zeit

ACTION a_Error:
Q_sError := '';

IF Q_bVorwarnungZeitintervall
THEN
	Q_sError := 'Bremsentest innerhalb der nächsten 15min nötig!';
END_IF

IF TO_UDINT(I_nDiagNummer) = cUberschreitungZeitBremsentest
THEN
	Q_sError := 'Bremsentest nötig! Fehler quittieren und Bremsentest ausführen';
END_IF

IF Q_bErr_Bremsoeffnung
	OR Q_bErr_Haltebremse
	OR Q_bErr_Haltemoment
THEN
	Q_sError := 'Fehler beim Bremsentest';
END_IF

IF Q_bErr_Bremsoeffnung
THEN
	Q_sError := CONCAT(Q_sError,'| Fehler Bremsöffnung');
END_IF

IF Q_bErr_Haltebremse
THEN
	Q_sError := CONCAT(Q_sError,'| Fehler Haltebremse');
END_IF

IF Q_bErr_Haltemoment
THEN
	Q_sError := CONCAT(Q_sError,'| Fehler Haltemoment');
END_IF

IF nFehlerZaehler <> 0
THEN
	Q_sError := CONCAT(Q_sError,'-> ');
	Q_sError := CONCAT(Q_sError,TO_STRING(10-nFehlerZaehler));
	Q_sError := CONCAT(Q_sError,' Versuche übrig!');
END_IF

IF Q_bFatalError
THEN
	Q_sError := 'Schutzbereich stillgelegt -> Bremsfunktion defekt!';
END_IF
END_ACTION

ACTION a_LogZeile:

Q_sLogZeile := '';
Q_sLogZeile	:= I_stZeitstempel.sTimeStamp;

IF Q_bErr_Haltebremse
THEN
	Q_sLogZeile:= CONCAT(Q_sLogZeile,'n.IO;');
ELSE
	Q_sLogZeile:= CONCAT(Q_sLogZeile,'IO;');
END_IF
IF Q_bErr_Bremsoeffnung
THEN
	Q_sLogZeile:= CONCAT(Q_sLogZeile,'n.IO;');
ELSE
	Q_sLogZeile:= CONCAT(Q_sLogZeile,'IO;');
END_IF
IF Q_bErr_Haltemoment
THEN
	Q_sLogZeile:= CONCAT(Q_sLogZeile,'n.IO;');
ELSE
	Q_sLogZeile:= CONCAT(Q_sLogZeile,'IO;');
END_IF
END_ACTION

END_FUNCTION_BLOCK

// POUs/FB_CtrlXGrupEinschalt
// Dieser FB schaltet die Zwischenkreisspannung für die Bosch CtrlX-Drive von dem Einspeisemodul auf die Slavemodule frei.
FUNCTION_BLOCK FB_CtrlXGrupEinschalt
VAR_IN_OUT
	IQ_arrAlleAchsen		: ARRAY [0..cAnzAchsen] OF TC3_UniLib.ST_NcAchsen;	// Schnittstelle zu allen Achsen
END_VAR
VAR_INPUT
	I_bNetzEin				: BOOL;	// Spannungsversorgung für die Servos zuschalten
	I_bQuittError			: BOOL;	// Quittiert alle Fehler und Wartet auf wiedereinschalten
	I_tAbschaltVerz		: TIME := T#1S;	// Abschaltzeit für die Servos
	I_nAxisIDEinspeisung	: INT;	//	Achs-ID für von dem Einspeise-Servo
	I_arrAxisIDSlave		: ARRAY [1..cAnzAchsen] OF INT;	// Achs-IDs der am Master (I_nAxisIDEinspeisung) angeschlossenen Wechselrichter-Servos
	I_nAnzahlSlaves		: INT;	// Anzahl der in I_arrAxisIDSlave angebundene Achsen
END_VAR
VAR_OUTPUT
	Q_bGruppeFrg			: ARRAY [1..TC3_UniLib.cAnzSchutzBer] OF BOOL;	// Schutzbereich geschlossen und Antriebe sind eingeschaltet
	Q_bGruppeFrgVerz		: ARRAY [1..TC3_UniLib.cAnzSchutzBer] OF BOOL;	// Schutzbereich geschlossen und Antriebe sind verzögert ausgeschaltet
	Q_bAntriebeEin			: BOOL;	// Alle Antriebe sind an
	Q_bAntriebeAus			: BOOL;	// Alle Antriebe sind aus
	Q_bGruppeError			: BOOL;	// Achs-Gruppe hat einen Error
	Q_sGruppeError			: STRING;	// Achs-Gruppen-Error als Klartext
END_VAR
VAR	
	nStep				: INT;
	nIdx				: INT;
	nFehler			: INT;
	tonTimer			: Tc2_Standard.TON;
	tofFrgVerz		: ARRAY [1..TC3_UniLib.cAnzSchutzBer] OF Tc2_Standard.TOF;
	nLastStep		: INT;
	bSlavesBb		: BOOL;
	bSlavesAF		: BOOL;
	bFrgVerzAus		: BOOL;
	bAntriebeEin	: BOOL;
	tonAntriebeAus	:Tc2_Standard.TON;
	tonGruppeFrgVerzAus	:Tc2_Standard.TON;
END_VAR

IF NOT I_bNetzEin
THEN
	bAntriebeEin	:= FALSE;
ELSIF I_bNetzEin
	AND Q_bAntriebeAus
THEN
	bAntriebeEin	:= TRUE;
END_IF

tonAntriebeAus(
	IN := NOT bAntriebeEin,
	PT := t#5s,
	Q => Q_bAntriebeAus); 
	
// Ermitteln, ob alle Salves Betriebsbereit sind
FOR nIdx := 1 TO I_nAnzahlSlaves DO
	IF IQ_arrAlleAchsen[I_arrAxisIDSlave[nIdx]].stEinAusG.I_nDCStatusword.0
	THEN
		bSlavesBb := TRUE;
	ELSE
		bSlavesBb := FALSE;
		EXIT;		
	END_IF
END_FOR

/////////////////////////////////////////////////////////////////////
//Schreiben des BtB in die Achsstrucktur
IQ_arrAlleAchsen[I_nAxisIDEinspeisung].stStatus.bAchseBTB 	:= IQ_arrAlleAchsen[I_nAxisIDEinspeisung].stEinAusG.I_nEinspeiseStatusword.15;

FOR nIdx := 1 TO LIMIT(1,I_nAnzahlSlaves,cAnzAchsen) DO
	IQ_arrAlleAchsen[I_arrAxisIDSlave[nIdx]].stStatus.bAchseBTB	:=
		IQ_arrAlleAchsen[I_arrAxisIDSlave[nIdx]].stEinAusG.I_nDCStatusword.0	// Status BB-Relais
		AND NOT IQ_arrAlleAchsen[I_arrAxisIDSlave[nIdx]].stEinAusG.I_nDCStatusword.13;	// Antriebs-Fehler
END_FOR 

CASE nStep OF
/////////////////////////////////////////////////////////////////////	
0: //INIT
	bSlavesAF 				:= FALSE;
	nFehler 					:= 0;
	Q_bGruppeError			:= FALSE;
	Q_bAntriebeEin			:= FALSE;
	Q_sGruppeError			:= '';
	FOR nIdx:= 1 TO LIMIT(1,I_nAnzahlSlaves,cAnzAchsen) DO	
		IQ_arrAlleAchsen[I_arrAxisIDSlave[nIdx]].stEinAusG.Q_nDCPowerControl.0 :=FALSE;
	END_FOR
	IQ_arrAlleAchsen[I_nAxisIDEinspeisung].stEinAusG.Q_nEinspeiseSteuerwort.15 := 
	IQ_arrAlleAchsen[I_nAxisIDEinspeisung].stEinAusG.Q_nEinspeiseSteuerwort.14 :=
	IQ_arrAlleAchsen[I_nAxisIDEinspeisung].stEinAusG.Q_nEinspeiseSteuerwort.12 := FALSE;
	FOR nIdx :=1 TO cAnzSchutzBer DO
		Q_bGruppeFrg[nIdx] 		:= FALSE;
		Q_bGruppeFrgVerz[nIdx] 	:= FALSE;
	END_FOR
	nStep 				:= 10;
	
/////////////////////////////////////////////////////////////////////	
10: //Warten auf Netzeinschaltung
	IF bAntriebeEin
	THEN
		nStep := 15;
	END_IF
/////////////////////////////////////////////////////////////////////	
15: //Warten auf Betriebsbereit der Salves
	IF bSlavesBb
	THEN
		nStep := 20;
	ELSIF tonTimer.Q
	THEN
		nFehler 	:= 10;
		nStep 	:= -100;
	END_IF
/////////////////////////////////////////////////////////////////////	
20: //Warten auf Hardware bereit zum Einschalten & Netzspannung OK
	IF IQ_arrAlleAchsen[I_nAxisIDEinspeisung].stEinAusG.I_nEinspeiseStatusword.4 // Netzspannung OK
		AND IQ_arrAlleAchsen[I_nAxisIDEinspeisung].stEinAusG.I_nEinspeiseStatusword.5 // Hardware bereit zum Einschalten
	THEN
		nStep := 30;
	ELSIF tonTimer.Q
		AND NOT IQ_arrAlleAchsen[I_nAxisIDEinspeisung].stEinAusG.I_nEinspeiseStatusword.4 // Netzspannung OK
	THEN
		nFehler 	:= 20;
		nStep 	:= -100;
	ELSIF tonTimer.Q
		AND NOT IQ_arrAlleAchsen[I_nAxisIDEinspeisung].stEinAusG.I_nEinspeiseStatusword.5 // Hardware bereit zum Einschalten
	THEN
		nFehler 	:= 21;
		nStep 	:= -100;
	END_IF	
/////////////////////////////////////////////////////////////////////	
30: //Zwischenkreis laden und Netzschütz einschalteten - Gerät geht in Gleichrichterbetrieb
	IQ_arrAlleAchsen[I_nAxisIDEinspeisung].stEinAusG.Q_nEinspeiseSteuerwort.12 :=
	IQ_arrAlleAchsen[I_nAxisIDEinspeisung].stEinAusG.Q_nEinspeiseSteuerwort.14 := TRUE;
	IF IQ_arrAlleAchsen[I_nAxisIDEinspeisung].stEinAusG.I_nEinspeiseStatusword.6
		AND IQ_arrAlleAchsen[I_nAxisIDEinspeisung].stEinAusG.I_nEinspeiseStatusword.14
	THEN
		nStep := 40;
	ELSIF tonTimer.Q
		AND NOT IQ_arrAlleAchsen[I_nAxisIDEinspeisung].stEinAusG.I_nEinspeiseStatusword.6
	THEN
		nFehler 	:= 30;
		nStep 	:= -100;
	ELSIF tonTimer.Q
		AND NOT IQ_arrAlleAchsen[I_nAxisIDEinspeisung].stEinAusG.I_nEinspeiseStatusword.14
	THEN
		nFehler 	:= 31;
		nStep 	:= -100;
	END_IF
/////////////////////////////////////////////////////////////////////	
40: //Wirkt auf die IGBT-Brücke des Versorgungsgeräts, aktiviert die DC-Zwischenkreisspannungsregelung und die Sollbetriebsart
	IQ_arrAlleAchsen[I_nAxisIDEinspeisung].stEinAusG.Q_nEinspeiseSteuerwort.15 := TRUE;
	IF IQ_arrAlleAchsen[I_nAxisIDEinspeisung].stEinAusG.I_nEinspeiseStatusword.15
	THEN
		nStep := 50;
	ELSIF tonTimer.Q
	THEN
		nFehler 	:= 40;
		nStep 	:= -100;
	END_IF
/////////////////////////////////////////////////////////////////////	
50: //Slaveantriebe in AF umschalten
	FOR nIdx:= 1 TO LIMIT(1,I_nAnzahlSlaves,cAnzAchsen) DO	
		IQ_arrAlleAchsen[I_arrAxisIDSlave[nIdx]].stEinAusG.Q_nDCPowerControl.0 :=TRUE;
	END_FOR
	nStep := 60;
	
/////////////////////////////////////////////////////////////////////	
60: //Warten auf Antriebe Aus	
	Q_bAntriebeEin	:= TRUE;
	FOR nIdx :=1 TO TC3_UniLib.cAnzSchutzBer DO
		tofFrgVerz[nIdx](	IN := arrSchutzEinrGeschl[nIdx],
								PT:= I_tAbschaltVerz);
		Q_bGruppeFrg[nIdx] 		:= arrSchutzEinrGeschl[nIdx];
		Q_bGruppeFrgVerz[nIdx] 	:= tofFrgVerz[nIdx].Q;
	END_FOR
	

	FOR nIdx :=1 TO TC3_UniLib.cAnzSchutzBer DO
		IF Q_bGruppeFrgVerz[nIdx]
		THEN
			bFrgVerzAus	 	:= FALSE;
			EXIT;
		ELSE
			bFrgVerzAus := TRUE;
		END_IF
	END_FOR
	
	tonGruppeFrgVerzAus(IN := bFrgVerzAus,
								PT:= t#5s);
	
	IF NOT bAntriebeEin
		AND tonGruppeFrgVerzAus.Q
	THEN
		bFrgVerzAus	 	:= FALSE;
		nStep 			:= 0;
	END_IF

/////////////////////////////////////////////////////////////////////	
-100: //Fehlerschritt
	Q_bGruppeError			:= TRUE;
	CASE nFehler OF
		10: Q_sGruppeError			:= 'Mindestens ein Regler meldet nicht betriebsbereit!';
		20: Q_sGruppeError			:= 'Netzspannung an der Einspeisung nicht OK!';
		21: Q_sGruppeError			:= 'Hardware nicht bereit zur Leistungszuschaltung!';
		30: Q_sGruppeError			:= 'Zwischenkreis ist nicht geladen, Thyristoren sind gesperrt!';
		31: Q_sGruppeError			:= 'Nicht bereit zur Freigabe: z.B. Netzschütz aus, Ladewiderstand aktiv!';
		40: Q_sGruppeError			:= 'Zwischenkreis nicht belastbar, Antriebsfreigabe darf nicht gesetzt werden!';
	END_CASE
	IF I_bQuittError
		OR NOT bAntriebeEin
	THEN
		nStep := 0;
	END_IF

END_CASE

tonTimer(IN:= (nStep = nLastStep),
			PT := t#15s); 
IF nStep <> nLastStep
THEN
	nLastStep := nStep;
END_IF

END_FUNCTION_BLOCK

// VISUs/Intern/V_DiagAchse
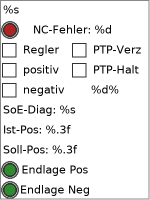
VISUALIZATION V_DiagAchse  // 150x200
// Diese Visu muss in einer anderen Übersichts-Visu aufgerufen werden. Sie ist nicht eigenständig.
VAR_INPUT
	I_stNcAchsen	: TC3_UniLib.ST_NcAchsen;
END_VAR
    Lamp1 (0,20 20x20), variable: I_stNcAchsen.bNcFehler, style: Lamp-Lamp1-Red
    Rectangle (30,20 120x20), "NC-Fehler: %d", text variable: I_stNcAchsen.nFehlerNr
    Checkbox (0,40 70x20), "Regler", variable: I_stNcAchsen.bBetrbBer, input disabled if: TRUE
    Rectangle (0,100 150x20), "SoE-Diag: %s", text variable: arrAchsDiag[I_stNcAchsen.nAxNr]
    Rectangle (0,0 150x20), "%s", text variable: I_stNcAchsen.sAxName
    Checkbox (0,60 70x20), "positiv", variable: I_stNcAchsen.stFreigb.bVorsFrgPos, input disabled if: TRUE
    Checkbox (0,80 70x20), "negativ", variable: I_stNcAchsen.stFreigb.bVorsFrgNeg, input disabled if: TRUE
    Rectangle (0,120 150x20), "Ist-Pos: %.3f", text variable: I_stNcAchsen.fPosIstwert
    Rectangle (0,140 150x20), "Soll-Pos: %.3f", text variable: I_stNcAchsen.stAuftrg.fPTP_ZielPos
    Checkbox (70,40 80x20), "PTP-Verz", variable: I_stNcAchsen.stAuftrg.bPTP_halt, input disabled if: TRUE
    Checkbox (70,60 80x20), "PTP-Halt", variable: I_stNcAchsen.stAuftrg.bPTP_halt, input disabled if: TRUE
    Lamp1 (0,160 20x20), variable: I_stNcAchsen.stFreigb.bSensEndlPos, style: Lamp-Lamp1-Green
    Lamp1 (0,180 20x20), variable: I_stNcAchsen.stFreigb.bSensEndlNeg, style: Lamp-Lamp1-Green
    Label (20,160 70x20), "Endlage Pos"
    Label (20,180 70x20), "Endlage Neg"
    Rectangle (70,80 70x20), "%d%", text variable: I_stNcAchsen.fAuftrOverride
END_VISUALIZATION
